KUKA KRL program: EPS_2_25716_MHDR08_A_20251212040354.src

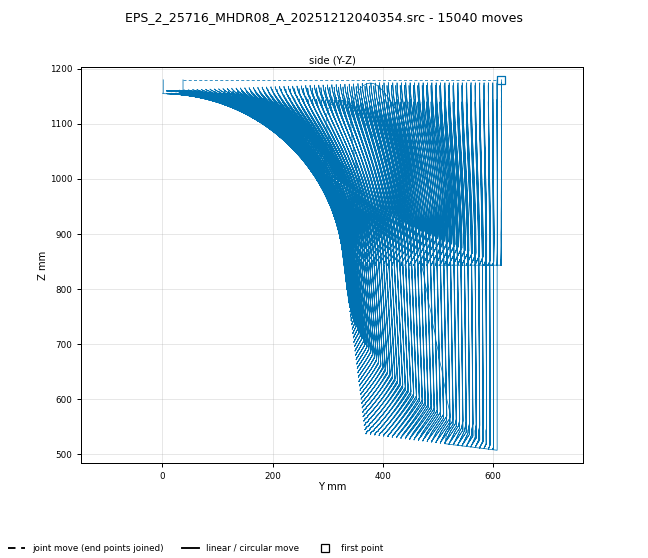
[picture p0: tool path of EPS_2_25716_MHDR08_A_20251212040354.src, 15040 of 15042 moves have a stored position in this frame; points joined in program order, loops and branches not executed]
&ACCESS RVP
&REL 4
&COMMENT QRS 19112012
&PARAM EDITMASK = *
DEF PART()
EXT BAS (BAS_COMMAND :IN,REAL :IN )
INT I
BAS (#INITMOV,0 )

;KUKA QRS Post kuka4.cps  Date:22-06-2017 !

File_ID=2954

QRS_PRE_INIT()

;Init var - Until changes are made in qrs_pre_init
Outlet_Square_prg=0
Inlet_1_Square_prg=0
Inlet_2_Square_prg=0
Inlet_3_Square_prg=0
Inlet_4_Square_prg=0
Inlet_5_Square_prg=0

Outlet_1={X 0.000, Y 400.000, Z 865.000, B 0.000, E1 0.000 }
Inlet_1={X 0.000, Y 400.000, Z 835.000, B 0.000, E1 180.000 }
Outlet_1_type=610
Inlet_1_type=610
;QRS#1=Sidecore dimensions
;QRS#2=600-24" Concrete
;QRS#3=600-24" Concrete
;QRS#4=
;QRS#5=
;QRS#6=
;QRS#7=
;QRS#8=
;QRS#9=S306-34L
;QRS#10=S306-34L
;QRS#11=
;QRS#12=
;QRS#13=
;QRS#14=
;QRS#15=
;QRS#16=1220x127x1524 5'
;QRS#17=EPS Height
;QRS#18=1170
;QRS#19=*
;QRS#20= UPDATED VERSION 22-06-2017
;QRS#21=*
Outlet_Square=0450
Inlet_1_Square=0450
Inlet_2_Square=0
Inlet_3_Square=0
Inlet_4_Square=0
Inlet_5_Square=0
Mill_Square=1
Outlet_Square_Prg=264
Inlet_1_Square_prg=264

QRS_INIT()

$ADVANCE=5

; T1
PTP {E1 172.54,E2 172.54}
PTP {X 0,Y 615.615,A -85,B 0,C 180,E1 172.54,E2 172.54,E3 0,E4 0,E5 0,E6 0}
QRS_SPEED_INIT()
LIN {X 0,Y 615.615,Z 1180,A -85,B 0,C 180,E1 172.54,E2 172.54,E3 0,E4 0,E5 0,E6 0} C_VEL
LIN {X 0,Y 615.615,Z 845.44,A -85,B 0,C 180,E1 172.54,E2 172.54} C_VEL
LIN {X 0,Y 615.56,Z 843.44,A -85,B 0,C 180,E1 172.726,E2 172.726} C_VEL
LIN {X 0,Y 615.848,Z 843.44,A -85,B 0,C 180,E1 176.52,E2 176.52} C_VEL
LIN {X 0,Y 615.869,Z 843.44,A -85,B 0,C 180,E1 181.159,E2 181.159} C_VEL
LIN {X 0,Y 615.847,Z 843.44,A -85,B 0,C 180,E1 185.807,E2 185.807} C_VEL
LIN {X 0,Y 615.82,Z 843.44,A -85,B 0,C 180,E1 190.493,E2 190.493} C_VEL
LIN {X 0,Y 615.8,Z 843.44,A -85,B 0,C 180,E1 195.252,E2 195.252} C_VEL
LIN {X 0,Y 615.797,Z 843.44,A -85,B 0,C 180,E1 200.122,E2 200.122} C_VEL
LIN {X 0,Y 615.751,Z 843.44,A -85,B 0,C 180,E1 205.15,E2 205.15} C_VEL
LIN {X 0,Y 615.231,Z 843.44,A -85,B 0,C 180,E1 207.766,E2 207.766} C_VEL
LIN {X 0,Y 615.751,Z 843.44,A -85,B 0,C 180,E1 210.394,E2 210.394} C_VEL
LIN {X 0,Y 615.134,Z 843.44,A -85,B 0,C 180,E1 213.842,E2 213.842} C_VEL
LIN {X 0,Y 615.66,Z 843.44,A -85,B 0,C 180,E1 215.943,E2 215.943} C_VEL
LIN {X 0,Y 615.4,Z 843.44,A -85,B 0,C 180,E1 217.841,E2 217.841} C_VEL
LIN {X 0,Y 615.353,Z 843.44,A -85,B 0,C 180,E1 218.886,E2 218.886} C_VEL
LIN {X 0,Y 615.632,Z 843.44,A -85,B 0,C 180,E1 221.501,E2 221.501} C_VEL
LIN {X 0,Y 615.673,Z 843.44,A -85,B 0,C 180,E1 225.106,E2 225.106} C_VEL
LIN {X 0,Y 615.248,Z 843.44,A -85,B 0,C 180,E1 228.539,E2 228.539} C_VEL
LIN {X 0,Y 615.62,Z 843.44,A -85,B 0,C 180,E1 231.134,E2 231.134} C_VEL
LIN {X 0,Y 615.854,Z 843.44,A -85,B 0,C 180,E1 236.479,E2 236.479} C_VEL
LIN {X 0,Y 615.651,Z 843.44,A -85,B 0,C 180,E1 236.67,E2 236.67} C_VEL
LIN {X 0,Y 615.102,Z 843.529,A -85,B 0,C 180,E1 236.769,E2 236.769} C_VEL
LIN {X 0,Y 615.262,Z 884.389,A -85,B 0,C 180,E1 237.344,E2 237.344} C_VEL
LIN {X 0,Y 615.454,Z 896.053,A -85,B 0,C 180,E1 237.545,E2 237.545} C_VEL
LIN {X 0,Y 615.368,Z 912.24,A -85,B 0,C 180,E1 237.89,E2 237.89} C_VEL
LIN {X 0,Y 615.486,Z 927.188,A -85,B 0,C 180,E1 238.298,E2 238.298} C_VEL
LIN {X 0,Y 615.404,Z 942.776,A -85,B 0,C 180,E1 238.798,E2 238.798} C_VEL
LIN {X 0,Y 615.565,Z 957.668,A -85,B 0,C 180,E1 239.371,E2 239.371} C_VEL
LIN {X 0,Y 615.586,Z 971.276,A -85,B 0,C 180,E1 239.959,E2 239.959} C_VEL
LIN {X 0,Y 615.496,Z 984.135,A -85,B 0,C 180,E1 240.573,E2 240.573} C_VEL
LIN {X 0,Y 615.632,Z 998.101,A -85,B 0,C 180,E1 241.333,E2 241.333} C_VEL
LIN {X 0,Y 615.649,Z 1011.417,A -85,B 0,C 180,E1 242.129,E2 242.129} C_VEL
LIN {X 0,Y 615.606,Z 1024.492,A -85,B 0,C 180,E1 242.987,E2 242.987} C_VEL
LIN {X 0,Y 615.637,Z 1037.892,A -85,B 0,C 180,E1 243.961,E2 243.961} C_VEL
LIN {X 0,Y 615.676,Z 1049.111,A -85,B 0,C 180,E1 244.847,E2 244.847} C_VEL
LIN {X 0,Y 615.679,Z 1060.739,A -85,B 0,C 180,E1 245.844,E2 245.844} C_VEL
LIN {X 0,Y 615.643,Z 1071.153,A -85,B 0,C 180,E1 246.809,E2 246.809} C_VEL
LIN {X 0,Y 615.684,Z 1081.458,A -85,B 0,C 180,E1 247.846,E2 247.846} C_VEL
LIN {X 0,Y 615.684,Z 1091.552,A -85,B 0,C 180,E1 248.945,E2 248.945} C_VEL
LIN {X 0,Y 615.6,Z 1100.745,A -85,B 0,C 180,E1 250.026,E2 250.026} C_VEL
LIN {X 0,Y 615.667,Z 1109.198,A -85,B 0,C 180,E1 251.104,E2 251.104} C_VEL
LIN {X 0,Y 615.76,Z 1116.662,A -85,B 0,C 180,E1 252.141,E2 252.141} C_VEL
LIN {X 0,Y 615.563,Z 1125.951,A -85,B 0,C 180,E1 253.537,E2 253.537} C_VEL
LIN {X 0,Y 615.67,Z 1133.147,A -85,B 0,C 180,E1 254.744,E2 254.744} C_VEL
LIN {X 0,Y 615.818,Z 1137.992,A -85,B 0,C 180,E1 255.648,E2 255.648} C_VEL
LIN {X 0,Y 615.63,Z 1142.571,A -85,B 0,C 180,E1 256.539,E2 256.539} C_VEL
LIN {X 0,Y 615.562,Z 1146.872,A -85,B 0,C 180,E1 257.431,E2 257.431} C_VEL
LIN {X 0,Y 615.799,Z 1153.082,A -85,B 0,C 180,E1 258.916,E2 258.916} C_VEL
LIN {X 0,Y 615.609,Z 1157.519,A -85,B 0,C 180,E1 260.092,E2 260.092} C_VEL
LIN {X 0,Y 615.522,Z 1161.322,A -85,B 0,C 180,E1 261.266,E2 261.266} C_VEL
LIN {X 0,Y 615.732,Z 1165.013,A -85,B 0,C 180,E1 262.603,E2 262.603} C_VEL
LIN {X 0,Y 615.726,Z 1166.643,A -85,B 0,C 180,E1 263.27,E2 263.27} C_VEL
LIN {X 0,Y 615.525,Z 1168.699,A -85,B 0,C 180,E1 264.19,E2 264.19} C_VEL
LIN {X 0,Y 615.498,Z 1171.145,A -85,B 0,C 180,E1 265.588,E2 265.588} C_VEL
LIN {X 0,Y 615.665,Z 1172.314,A -85,B 0,C 180,E1 266.519,E2 266.519} C_VEL
LIN {X 0,Y 615.731,Z 1173.295,A -85,B 0,C 180,E1 267.448,E2 267.448} C_VEL
LIN {X 0,Y 615.468,Z 1174.226,A -85,B 0,C 180,E1 268.84,E2 268.84} C_VEL
LIN {X 0,Y 615.846,Z 1174.153,A -85,B 0,C 180,E1 271.159,E2 271.159} C_VEL
LIN {X 0,Y 615.739,Z 1173.293,A -85,B 0,C 180,E1 272.552,E2 272.552} C_VEL
LIN {X 0,Y 615.821,Z 1172.284,A -85,B 0,C 180,E1 273.48,E2 273.48} C_VEL
LIN {X 0,Y 615.545,Z 1170.345,A -85,B 0,C 180,E1 274.878,E2 274.878} C_VEL
LIN {X 0,Y 615.53,Z 1168.698,A -85,B 0,C 180,E1 275.81,E2 275.81} C_VEL
LIN {X 0,Y 615.68,Z 1166.586,A -85,B 0,C 180,E1 276.76,E2 276.76} C_VEL
LIN {X 0,Y 615.774,Z 1164.622,A -85,B 0,C 180,E1 277.538,E2 277.538} C_VEL
LIN {X 0,Y 615.541,Z 1161.319,A -85,B 0,C 180,E1 278.733,E2 278.733} C_VEL
LIN {X 0,Y 615.557,Z 1157.527,A -85,B 0,C 180,E1 279.908,E2 279.908} C_VEL
LIN {X 0,Y 615.815,Z 1153.08,A -85,B 0,C 180,E1 281.083,E2 281.083} C_VEL
LIN {X 0,Y 615.534,Z 1146.875,A -85,B 0,C 180,E1 282.57,E2 282.57} C_VEL
LIN {X 0,Y 615.601,Z 1139.632,A -85,B 0,C 180,E1 284.058,E2 284.058} C_VEL
LIN {X 0,Y 615.808,Z 1133.136,A -85,B 0,C 180,E1 285.252,E2 285.252} C_VEL
LIN {X 0,Y 615.58,Z 1124.652,A -85,B 0,C 180,E1 286.664,E2 286.664} C_VEL
LIN {X 0,Y 615.672,Z 1115.983,A -85,B 0,C 180,E1 287.956,E2 287.956} C_VEL
LIN {X 0,Y 615.786,Z 1109.198,A -85,B 0,C 180,E1 288.892,E2 288.892} C_VEL
LIN {X 0,Y 615.593,Z 1098.188,A -85,B 0,C 180,E1 290.283,E2 290.283} C_VEL
LIN {X 0,Y 615.645,Z 1088.781,A -85,B 0,C 180,E1 291.367,E2 291.367} C_VEL
LIN {X 0,Y 615.705,Z 1078.314,A -85,B 0,C 180,E1 292.476,E2 292.476} C_VEL
LIN {X 0,Y 615.619,Z 1068.945,A -85,B 0,C 180,E1 293.404,E2 293.404} C_VEL
LIN {X 0,Y 615.634,Z 1057.804,A -85,B 0,C 180,E1 294.418,E2 294.418} C_VEL
LIN {X 0,Y 615.649,Z 1046.141,A -85,B 0,C 180,E1 295.395,E2 295.395} C_VEL
LIN {X 0,Y 615.633,Z 1033.557,A -85,B 0,C 180,E1 296.362,E2 296.362} C_VEL
LIN {X 0,Y 615.629,Z 1022.093,A -85,B 0,C 180,E1 297.174,E2 297.174} C_VEL
LIN {X 0,Y 615.569,Z 1009.608,A -85,B 0,C 180,E1 297.987,E2 297.987} C_VEL
LIN {X 0,Y 615.637,Z 995.015,A -85,B 0,C 180,E1 298.837,E2 298.837} C_VEL
LIN {X 0,Y 615.587,Z 981.265,A -85,B 0,C 180,E1 299.562,E2 299.562} C_VEL
LIN {X 0,Y 615.487,Z 970.325,A -85,B 0,C 180,E1 300.092,E2 300.092} C_VEL
LIN {X 0,Y 615.592,Z 953.964,A -85,B 0,C 180,E1 300.777,E2 300.777} C_VEL
LIN {X 0,Y 615.412,Z 938.367,A -85,B 0,C 180,E1 301.352,E2 301.352} C_VEL
LIN {X 0,Y 615.482,Z 928.614,A -85,B 0,C 180,E1 301.657,E2 301.657} C_VEL
LIN {X 0,Y 615.497,Z 912.307,A -85,B 0,C 180,E1 302.101,E2 302.101} C_VEL
LIN {X 0,Y 615.3,Z 902.116,A -85,B 0,C 180,E1 302.336,E2 302.336} C_VEL
LIN {X 0,Y 615.425,Z 894.144,A -85,B 0,C 180,E1 302.489,E2 302.489} C_VEL
LIN {X 0,Y 615.395,Z 875.759,A -85,B 0,C 180,E1 302.773,E2 302.773} C_VEL
LIN {X 0,Y 615.134,Z 843.44,A -85,B 0,C 180,E1 303.235,E2 303.235} C_VEL
LIN {X 0,Y 615.646,Z 843.44,A -85,B 0,C 180,E1 303.33,E2 303.33} C_VEL
LIN {X 0,Y 615.853,Z 843.44,A -85,B 0,C 180,E1 303.52,E2 303.52} C_VEL
LIN {X 0,Y 615.62,Z 843.44,A -85,B 0,C 180,E1 308.866,E2 308.866} C_VEL
LIN {X 0,Y 615.242,Z 843.44,A -85,B 0,C 180,E1 311.943,E2 311.943} C_VEL
LIN {X 0,Y 615.68,Z 843.44,A -85,B 0,C 180,E1 314.895,E2 314.895} C_VEL
LIN {X 0,Y 615.622,Z 843.44,A -85,B 0,C 180,E1 318.499,E2 318.499} C_VEL
LIN {X 0,Y 615.342,Z 843.44,A -85,B 0,C 180,E1 321.113,E2 321.113} C_VEL
LIN {X 0,Y 615.398,Z 843.44,A -85,B 0,C 180,E1 322.159,E2 322.159} C_VEL
LIN {X 0,Y 615.655,Z 843.44,A -85,B 0,C 180,E1 324.057,E2 324.057} C_VEL
LIN {X 0,Y 615.136,Z 843.44,A -85,B 0,C 180,E1 326.841,E2 326.841} C_VEL
LIN {X 0,Y 615.745,Z 843.44,A -85,B 0,C 180,E1 329.606,E2 329.606} C_VEL
LIN {X 0,Y 615.22,Z 843.44,A -85,B 0,C 180,E1 332.234,E2 332.234} C_VEL
LIN {X 0,Y 615.744,Z 843.44,A -85,B 0,C 180,E1 334.85,E2 334.85} C_VEL
LIN {X 0,Y 615.807,Z 843.44,A -85,B 0,C 180,E1 339.879,E2 339.879} C_VEL
LIN {X 0,Y 615.814,Z 843.44,A -85,B 0,C 180,E1 343.784,E2 343.784} C_VEL
LIN {X 0,Y 615.822,Z 843.44,A -85,B 0,C 180,E1 349.507,E2 349.507} C_VEL
LIN {X 0,Y 615.852,Z 843.44,A -85,B 0,C 180,E1 354.193,E2 354.193} C_VEL
LIN {X 0,Y 615.873,Z 843.44,A -85,B 0,C 180,E1 358.841,E2 358.841} C_VEL
LIN {X 0,Y 615.858,Z 843.44,A -85,B 0,C 180,E1 363.48,E2 363.48} C_VEL
LIN {X 0,Y 615.852,Z 843.44,A -85,B 0,C 180,E1 368.143,E2 368.143} C_VEL
LIN {X 0,Y 615.792,Z 843.44,A -85,B 0,C 180,E1 372.862,E2 372.862} C_VEL
LIN {X 0,Y 615.794,Z 843.44,A -85,B 0,C 180,E1 377.671,E2 377.671} C_VEL
LIN {X 0,Y 615.796,Z 843.44,A -85,B 0,C 180,E1 377.992,E2 377.992} C_VEL
LIN {X 0,Y 615.771,Z 843.44,A -85,B 0,C 180,E1 382.613,E2 382.613} C_VEL
LIN {X 0,Y 615.222,Z 843.44,A -85,B 0,C 180,E1 385.173,E2 385.173} C_VEL
LIN {X 0,Y 615.721,Z 843.44,A -85,B 0,C 180,E1 387.742,E2 387.742} C_VEL
LIN {X 0,Y 615.236,Z 843.44,A -85,B 0,C 180,E1 390.422,E2 390.422} C_VEL
LIN {X 0,Y 615.867,Z 843.44,A -85,B 0,C 180,E1 393.115,E2 393.115} C_VEL
LIN {X 0,Y 615.552,Z 843.44,A -85,B 0,C 180,E1 395.95,E2 395.95} C_VEL
LIN {X 0,Y 615.615,Z 843.44,A -85,B 0,C 180,E1 397.867,E2 397.867} C_VEL
LIN {X 0,Y 615.605,Z 843.44,A -85,B 0,C 180,E1 401.913,E2 401.913} C_VEL
LIN {X 0,Y 615.188,Z 843.44,A -85,B 0,C 180,E1 405.151,E2 405.151} C_VEL
LIN {X 0,Y 615.672,Z 843.44,A -85,B 0,C 180,E1 408.093,E2 408.093} C_VEL
LIN {X 0,Y 615.538,Z 843.44,A -85,B 0,C 180,E1 412.143,E2 412.143} C_VEL
LIN {X 0,Y 615.49,Z 843.44,A -85,B 0,C 180,E1 414.046,E2 414.046} C_VEL
LIN {X 0,Y 615.859,Z 843.44,A -85,B 0,C 180,E1 416.885,E2 416.885} C_VEL
LIN {X 0,Y 615.114,Z 843.44,A -85,B 0,C 180,E1 417.064,E2 417.064} C_VEL
LIN {X 0,Y 614.862,Z 846.621,A -85,B 0,C 180,E1 417.161,E2 417.161} C_VEL
LIN {X 0,Y 615.416,Z 866.536,A -85,B 0,C 180,E1 417.507,E2 417.507} C_VEL
LIN {X 0,Y 615.402,Z 882.125,A -85,B 0,C 180,E1 417.844,E2 417.844} C_VEL
LIN {X 0,Y 615.386,Z 891.155,A -85,B 0,C 180,E1 418.082,E2 418.082} C_VEL
LIN {X 0,Y 615.464,Z 900.26,A -85,B 0,C 180,E1 418.35,E2 418.35} C_VEL
LIN {X 0,Y 615.435,Z 912.408,A -85,B 0,C 180,E1 418.742,E2 418.742} C_VEL
LIN {X 0,Y 615.43,Z 919.467,A -85,B 0,C 180,E1 419.003,E2 419.003} C_VEL
LIN {X 0,Y 615.562,Z 927.899,A -85,B 0,C 180,E1 419.336,E2 419.336} C_VEL
LIN {X 0,Y 615.593,Z 942.209,A -85,B 0,C 180,E1 419.959,E2 419.959} C_VEL
LIN {X 0,Y 615.496,Z 955.26,A -85,B 0,C 180,E1 420.588,E2 420.588} C_VEL
LIN {X 0,Y 615.62,Z 968.859,A -85,B 0,C 180,E1 421.332,E2 421.332} C_VEL
LIN {X 0,Y 615.633,Z 982.469,A -85,B 0,C 180,E1 422.152,E2 422.152} C_VEL
LIN {X 0,Y 615.603,Z 995.12,A -85,B 0,C 180,E1 422.987,E2 422.987} C_VEL
LIN {X 0,Y 615.636,Z 1007.438,A -85,B 0,C 180,E1 423.88,E2 423.88} C_VEL
LIN {X 0,Y 615.669,Z 1019.641,A -85,B 0,C 180,E1 424.846,E2 424.846} C_VEL
LIN {X 0,Y 615.679,Z 1030.462,A -85,B 0,C 180,E1 425.774,E2 425.774} C_VEL
LIN {X 0,Y 615.64,Z 1041.606,A -85,B 0,C 180,E1 426.809,E2 426.809} C_VEL
LIN {X 0,Y 615.688,Z 1051.876,A -85,B 0,C 180,E1 427.846,E2 427.846} C_VEL
LIN {X 0,Y 615.697,Z 1061.937,A -85,B 0,C 180,E1 428.946,E2 428.946} C_VEL
LIN {X 0,Y 615.595,Z 1071.099,A -85,B 0,C 180,E1 430.026,E2 430.026} C_VEL
LIN {X 0,Y 615.667,Z 1079.523,A -85,B 0,C 180,E1 431.104,E2 431.104} C_VEL
LIN {X 0,Y 615.764,Z 1086.985,A -85,B 0,C 180,E1 432.14,E2 432.14} C_VEL
LIN {X 0,Y 615.566,Z 1096.22,A -85,B 0,C 180,E1 433.537,E2 433.537} C_VEL
LIN {X 0,Y 615.668,Z 1103.4,A -85,B 0,C 180,E1 434.745,E2 434.745} C_VEL
LIN {X 0,Y 615.804,Z 1108.238,A -85,B 0,C 180,E1 435.647,E2 435.647} C_VEL
LIN {X 0,Y 615.627,Z 1112.789,A -85,B 0,C 180,E1 436.539,E2 436.539} C_VEL
LIN {X 0,Y 615.572,Z 1117.063,A -85,B 0,C 180,E1 437.431,E2 437.431} C_VEL
LIN {X 0,Y 615.796,Z 1123.25,A -85,B 0,C 180,E1 438.916,E2 438.916} C_VEL
LIN {X 0,Y 615.603,Z 1127.679,A -85,B 0,C 180,E1 440.092,E2 440.092} C_VEL
LIN {X 0,Y 615.518,Z 1131.468,A -85,B 0,C 180,E1 441.266,E2 441.266} C_VEL
LIN {X 0,Y 615.724,Z 1135.152,A -85,B 0,C 180,E1 442.608,E2 442.608} C_VEL
LIN {X 0,Y 615.727,Z 1136.74,A -85,B 0,C 180,E1 443.27,E2 443.27} C_VEL
LIN {X 0,Y 615.523,Z 1138.799,A -85,B 0,C 180,E1 444.19,E2 444.19} C_VEL
LIN {X 0,Y 615.453,Z 1140.437,A -85,B 0,C 180,E1 445.122,E2 445.122} C_VEL
LIN {X 0,Y 615.677,Z 1142.366,A -85,B 0,C 180,E1 446.519,E2 446.519} C_VEL
LIN {X 0,Y 615.732,Z 1143.326,A -85,B 0,C 180,E1 447.448,E2 447.448} C_VEL
LIN {X 0,Y 615.483,Z 1144.233,A -85,B 0,C 180,E1 448.84,E2 448.84} C_VEL
LIN {X 0,Y 615.843,Z 1144.144,A -85,B 0,C 180,E1 451.159,E2 451.159} C_VEL
LIN {X 0,Y 615.568,Z 1143.294,A -85,B 0,C 180,E1 452.553,E2 452.553} C_VEL
LIN {X 0,Y 615.557,Z 1142.28,A -85,B 0,C 180,E1 453.482,E2 453.482} C_VEL
LIN {X 0,Y 615.709,Z 1141.029,A -85,B 0,C 180,E1 454.411,E2 454.411} C_VEL
LIN {X 0,Y 615.761,Z 1139.446,A -85,B 0,C 180,E1 455.342,E2 455.342} C_VEL
LIN {X 0,Y 615.543,Z 1136.711,A -85,B 0,C 180,E1 456.67,E2 456.67} C_VEL
LIN {X 0,Y 615.605,Z 1133.938,A -85,B 0,C 180,E1 457.76,E2 457.76} C_VEL
LIN {X 0,Y 615.822,Z 1131.13,A -85,B 0,C 180,E1 458.729,E2 458.729} C_VEL
LIN {X 0,Y 615.588,Z 1127.355,A -85,B 0,C 180,E1 459.908,E2 459.908} C_VEL
LIN {X 0,Y 615.554,Z 1121.749,A -85,B 0,C 180,E1 461.384,E2 461.384} C_VEL
LIN {X 0,Y 615.808,Z 1116.642,A -85,B 0,C 180,E1 462.564,E2 462.564} C_VEL
LIN {X 0,Y 615.577,Z 1109.39,A -85,B 0,C 180,E1 464.059,E2 464.059} C_VEL
LIN {X 0,Y 615.62,Z 1102.887,A -85,B 0,C 180,E1 465.257,E2 465.257} C_VEL
LIN {X 0,Y 615.803,Z 1095.663,A -85,B 0,C 180,E1 466.456,E2 466.456} C_VEL
LIN {X 0,Y 615.584,Z 1087.681,A -85,B 0,C 180,E1 467.677,E2 467.677} C_VEL
LIN {X 0,Y 615.634,Z 1077.663,A -85,B 0,C 180,E1 469.05,E2 469.05} C_VEL
LIN {X 0,Y 615.76,Z 1069.127,A -85,B 0,C 180,E1 470.123,E2 470.123} C_VEL
LIN {X 0,Y 615.624,Z 1058.361,A -85,B 0,C 180,E1 471.368,E2 471.368} C_VEL
LIN {X 0,Y 615.652,Z 1049.313,A -85,B 0,C 180,E1 472.334,E2 472.334} C_VEL
LIN {X 0,Y 615.703,Z 1038.425,A -85,B 0,C 180,E1 473.403,E2 473.403} C_VEL
LIN {X 0,Y 615.653,Z 1027.2,A -85,B 0,C 180,E1 474.423,E2 474.423} C_VEL
LIN {X 0,Y 615.64,Z 1015.562,A -85,B 0,C 180,E1 475.395,E2 475.395} C_VEL
LIN {X 0,Y 615.649,Z 1004.057,A -85,B 0,C 180,E1 476.281,E2 476.281} C_VEL
LIN {X 0,Y 615.649,Z 991.401,A -85,B 0,C 180,E1 477.174,E2 477.174} C_VEL
LIN {X 0,Y 615.626,Z 978.933,A -85,B 0,C 180,E1 477.98,E2 477.98} C_VEL
LIN {X 0,Y 615.59,Z 967.05,A -85,B 0,C 180,E1 478.685,E2 478.685} C_VEL
LIN {X 0,Y 615.616,Z 951.527,A -85,B 0,C 180,E1 479.503,E2 479.503} C_VEL
LIN {X 0,Y 615.48,Z 938.091,A -85,B 0,C 180,E1 480.146,E2 480.146} C_VEL
LIN {X 0,Y 615.584,Z 924.036,A -85,B 0,C 180,E1 480.73,E2 480.73} C_VEL
LIN {X 0,Y 615.577,Z 908.655,A -85,B 0,C 180,E1 481.288,E2 481.288} C_VEL
LIN {X 0,Y 615.335,Z 894.951,A -85,B 0,C 180,E1 481.731,E2 481.731} C_VEL
LIN {X 0,Y 615.584,Z 879.877,A -85,B 0,C 180,E1 482.109,E2 482.109} C_VEL
LIN {X 0,Y 615.542,Z 864.831,A -85,B 0,C 180,E1 482.426,E2 482.426} C_VEL
LIN {X 0,Y 615.35,Z 855.68,A -85,B 0,C 180,E1 482.585,E2 482.585} C_VEL
LIN {X 0,Y 614.951,Z 848.797,A -85,B 0,C 180,E1 482.714,E2 482.714} C_VEL
LIN {X 0,Y 614.443,Z 845.073,A -85,B 0,C 180,E1 482.795,E2 482.795} C_VEL
LIN {X 0,Y 614.72,Z 843.44,A -85,B 0,C 180,E1 482.88,E2 482.88} C_VEL
LIN {X 0,Y 615.865,Z 843.44,A -85,B 0,C 180,E1 483.115,E2 483.115} C_VEL
LIN {X 0,Y 615.646,Z 843.44,A -85,B 0,C 180,E1 483.913,E2 483.913} C_VEL
LIN {X 0,Y 615.593,Z 843.44,A -85,B 0,C 180,E1 488.868,E2 488.868} C_VEL
LIN {X 0,Y 615.221,Z 843.44,A -85,B 0,C 180,E1 491.945,E2 491.945} C_VEL
LIN {X 0,Y 615.662,Z 843.44,A -85,B 0,C 180,E1 494.893,E2 494.893} C_VEL
LIN {X 0,Y 615.623,Z 843.44,A -85,B 0,C 180,E1 498.499,E2 498.499} C_VEL
LIN {X 0,Y 615.338,Z 843.44,A -85,B 0,C 180,E1 501.113,E2 501.113} C_VEL
LIN {X 0,Y 615.38,Z 843.44,A -85,B 0,C 180,E1 502.162,E2 502.162} C_VEL
LIN {X 0,Y 615.647,Z 843.44,A -85,B 0,C 180,E1 504.056,E2 504.056} C_VEL
LIN {X 0,Y 615.135,Z 843.44,A -85,B 0,C 180,E1 506.841,E2 506.841} C_VEL
LIN {X 0,Y 615.75,Z 843.44,A -85,B 0,C 180,E1 509.606,E2 509.606} C_VEL
LIN {X 0,Y 615.222,Z 843.44,A -85,B 0,C 180,E1 512.234,E2 512.234} C_VEL
LIN {X 0,Y 615.735,Z 843.44,A -85,B 0,C 180,E1 514.849,E2 514.849} C_VEL
LIN {X 0,Y 615.818,Z 843.44,A -85,B 0,C 180,E1 519.879,E2 519.879} C_VEL
LIN {X 0,Y 615.53,Z 843.44,A -85,B 0,C 180,E1 522.322,E2 522.322} C_VEL
LIN {X 0,Y 615.632,Z 843.44,A -85,B 0,C 180,E1 524.743,E2 524.743} C_VEL
LIN {X 0,Y 615.802,Z 843.44,A -85,B 0,C 180,E1 527.138,E2 527.138} C_VEL
LIN {X 0,Y 615.859,Z 843.44,A -85,B 0,C 180,E1 531.857,E2 531.857} C_VEL
LIN {X 0,Y 615.56,Z 843.44,A -85,B 0,C 180,E1 532.726,E2 532.726} C_VEL
LIN {X 0,Y 611.541,Z 843.44,A -85,B 0,C 180,E1 534.313,E2 534.313} C_VEL
LIN {X 0,Y 607.674,Z 843.44,A -85,B 0,C 180,E1 535.921,E2 535.921} C_VEL
LIN {X 0,Y 607.881,Z 843.44,A -85,B 0,C 180,E1 541.423,E2 541.423} C_VEL
LIN {X 0,Y 607.65,Z 843.44,A -85,B 0,C 180,E1 546.615,E2 546.615} C_VEL
LIN {X 0,Y 607.601,Z 843.44,A -85,B 0,C 180,E1 551.46,E2 551.46} C_VEL
LIN {X 0,Y 607.656,Z 843.44,A -85,B 0,C 180,E1 555.852,E2 555.852} C_VEL
LIN {X 0,Y 607.803,Z 843.44,A -85,B 0,C 180,E1 560.339,E2 560.339} C_VEL
LIN {X 0,Y 607.775,Z 843.44,A -85,B 0,C 180,E1 564.965,E2 564.965} C_VEL
LIN {X 0,Y 607.621,Z 843.44,A -85,B 0,C 180,E1 569.78,E2 569.78} C_VEL
LIN {X 0,Y 607.6,Z 843.44,A -85,B 0,C 180,E1 576.586,E2 576.586} C_VEL
LIN {X 0,Y 607.592,Z 843.44,A -85,B 0,C 180,E1 582.109,E2 582.109} C_VEL
LIN {X 0,Y 607.447,Z 843.44,A -85,B 0,C 180,E1 586.087,E2 586.087} C_VEL
LIN {X 0,Y 607.547,Z 843.44,A -85,B 0,C 180,E1 591.615,E2 591.615} C_VEL
LIN {X 0,Y 607.882,Z 843.44,A -85,B 0,C 180,E1 596.309,E2 596.309} C_VEL
LIN {X 0,Y 608.694,Z 910.185,A -85,B 0,C 180,E1 597.444,E2 597.444} C_VEL
LIN {X 0,Y 608.624,Z 952.563,A -85,B 0,C 180,E1 598.779,E2 598.779} C_VEL
LIN {X 0,Y 608.455,Z 992.837,A -85,B 0,C 180,E1 600.672,E2 600.672} C_VEL
LIN {X 0,Y 608.284,Z 1030.382,A -85,B 0,C 180,E1 603.064,E2 603.064} C_VEL
LIN {X 0,Y 608.152,Z 1064.017,A -85,B 0,C 180,E1 605.832,E2 605.832} C_VEL
LIN {X 0,Y 608.002,Z 1093.584,A -85,B 0,C 180,E1 608.907,E2 608.907} C_VEL
LIN {X 0,Y 607.946,Z 1119.324,A -85,B 0,C 180,E1 612.298,E2 612.298} C_VEL
LIN {X 0,Y 607.917,Z 1140.95,A -85,B 0,C 180,E1 615.994,E2 615.994} C_VEL
LIN {X 0,Y 607.762,Z 1157.905,A -85,B 0,C 180,E1 619.991,E2 619.991} C_VEL
LIN {X 0,Y 607.765,Z 1167.962,A -85,B 0,C 180,E1 623.584,E2 623.584} C_VEL
LIN {X 0,Y 607.833,Z 1173.637,A -85,B 0,C 180,E1 627.154,E2 627.154} C_VEL
LIN {X 0,Y 607.927,Z 1174.659,A -85,B 0,C 180,E1 631.423,E2 631.423} C_VEL
LIN {X 0,Y 607.66,Z 1170.729,A -85,B 0,C 180,E1 634.986,E2 634.986} C_VEL
LIN {X 0,Y 607.708,Z 1162.531,A -85,B 0,C 180,E1 638.568,E2 638.568} C_VEL
LIN {X 0,Y 607.717,Z 1149.388,A -85,B 0,C 180,E1 642.185,E2 642.185} C_VEL
LIN {X 0,Y 607.894,Z 1130.904,A -85,B 0,C 180,E1 645.847,E2 645.847} C_VEL
LIN {X 0,Y 607.971,Z 1107.131,A -85,B 0,C 180,E1 649.414,E2 649.414} C_VEL
LIN {X 0,Y 608.103,Z 1077.903,A -85,B 0,C 180,E1 652.814,E2 652.814} C_VEL
LIN {X 0,Y 608.241,Z 1044.822,A -85,B 0,C 180,E1 655.831,E2 655.831} C_VEL
LIN {X 0,Y 608.39,Z 1008.415,A -85,B 0,C 180,E1 658.419,E2 658.419} C_VEL
LIN {X 0,Y 608.572,Z 967.8,A -85,B 0,C 180,E1 660.583,E2 660.583} C_VEL
LIN {X 0,Y 608.756,Z 925.8,A -85,B 0,C 180,E1 662.137,E2 662.137} C_VEL
LIN {X 0,Y 608.78,Z 887.562,A -85,B 0,C 180,E1 662.996,E2 662.996} C_VEL
LIN {X 0,Y 607.881,Z 843.44,A -85,B 0,C 180,E1 663.693,E2 663.693} C_VEL
LIN {X 0,Y 607.456,Z 843.44,A -85,B 0,C 180,E1 669.641,E2 669.641} C_VEL
LIN {X 0,Y 607.521,Z 843.44,A -85,B 0,C 180,E1 675.936,E2 675.936} C_VEL
LIN {X 0,Y 607.417,Z 843.44,A -85,B 0,C 180,E1 680.366,E2 680.366} C_VEL
LIN {X 0,Y 607.4,Z 843.44,A -85,B 0,C 180,E1 685.153,E2 685.153} C_VEL
LIN {X 0,Y 607.567,Z 843.44,A -85,B 0,C 180,E1 690.377,E2 690.377} C_VEL
LIN {X 0,Y 607.782,Z 843.44,A -85,B 0,C 180,E1 695.035,E2 695.035} C_VEL
LIN {X 0,Y 607.676,Z 843.44,A -85,B 0,C 180,E1 700.672,E2 700.672} C_VEL
LIN {X 0,Y 607.276,Z 843.44,A -85,B 0,C 180,E1 705.612,E2 705.612} C_VEL
LIN {X 0,Y 607.749,Z 843.44,A -85,B 0,C 180,E1 709.991,E2 709.991} C_VEL
LIN {X 0,Y 607.925,Z 843.44,A -85,B 0,C 180,E1 714.302,E2 714.302} C_VEL
LIN {X 0,Y 607.59,Z 843.44,A -85,B 0,C 180,E1 720,E2 720} C_VEL
LIN {X 0,Y 607.669,Z 843.44,A -85,B 0,C 180,E1 724.272,E2 724.272} C_VEL
LIN {X 0,Y 607.799,Z 843.44,A -85,B 0,C 180,E1 728.566,E2 728.566} C_VEL
LIN {X 0,Y 607.865,Z 843.44,A -85,B 0,C 180,E1 732.91,E2 732.91} C_VEL
LIN {X 0,Y 607.592,Z 843.44,A -85,B 0,C 180,E1 738.836,E2 738.836} C_VEL
LIN {X 0,Y 607.584,Z 843.44,A -85,B 0,C 180,E1 743.413,E2 743.413} C_VEL
LIN {X 0,Y 607.668,Z 843.44,A -85,B 0,C 180,E1 748.151,E2 748.151} C_VEL
LIN {X 0,Y 607.956,Z 843.44,A -85,B 0,C 180,E1 753.096,E2 753.096} C_VEL
LIN {X 0,Y 607.561,Z 843.44,A -85,B 0,C 180,E1 758.382,E2 758.382} C_VEL
LIN {X 0,Y 607.634,Z 843.44,A -85,B 0,C 180,E1 762.105,E2 762.105} C_VEL
LIN {X 0,Y 607.753,Z 843.44,A -85,B 0,C 180,E1 768.146,E2 768.146} C_VEL
LIN {X 0,Y 607.557,Z 843.44,A -85,B 0,C 180,E1 773.409,E2 773.409} C_VEL
LIN {X 0,Y 607.902,Z 843.44,A -85,B 0,C 180,E1 776.687,E2 776.687} C_VEL
LIN {X 0,Y 608.629,Z 889.434,A -85,B 0,C 180,E1 777.639,E2 777.639} C_VEL
LIN {X 0,Y 608.621,Z 928.772,A -85,B 0,C 180,E1 778.986,E2 778.986} C_VEL
LIN {X 0,Y 608.5,Z 967.382,A -85,B 0,C 180,E1 780.877,E2 780.877} C_VEL
LIN {X 0,Y 608.281,Z 1006.644,A -85,B 0,C 180,E1 783.478,E2 783.478} C_VEL
LIN {X 0,Y 608.106,Z 1040.694,A -85,B 0,C 180,E1 786.413,E2 786.413} C_VEL
LIN {X 0,Y 607.909,Z 1070.334,A -85,B 0,C 180,E1 789.664,E2 789.664} C_VEL
LIN {X 0,Y 607.792,Z 1095.675,A -85,B 0,C 180,E1 793.224,E2 793.224} C_VEL
LIN {X 0,Y 607.753,Z 1114.665,A -85,B 0,C 180,E1 796.722,E2 796.722} C_VEL
LIN {X 0,Y 607.705,Z 1129.227,A -85,B 0,C 180,E1 800.351,E2 800.351} C_VEL
LIN {X 0,Y 607.76,Z 1138.059,A -85,B 0,C 180,E1 803.584,E2 803.584} C_VEL
LIN {X 0,Y 607.844,Z 1143.679,A -85,B 0,C 180,E1 807.154,E2 807.154} C_VEL
LIN {X 0,Y 607.892,Z 1144.632,A -85,B 0,C 180,E1 811.422,E2 811.422} C_VEL
LIN {X 0,Y 607.833,Z 1139.424,A -85,B 0,C 180,E1 815.699,E2 815.699} C_VEL
LIN {X 0,Y 607.755,Z 1128.941,A -85,B 0,C 180,E1 819.648,E2 819.648} C_VEL
LIN {X 0,Y 607.83,Z 1114.235,A -85,B 0,C 180,E1 823.276,E2 823.276} C_VEL
LIN {X 0,Y 607.912,Z 1093.883,A -85,B 0,C 180,E1 826.958,E2 826.958} C_VEL
LIN {X 0,Y 608.023,Z 1068.024,A -85,B 0,C 180,E1 830.521,E2 830.521} C_VEL
LIN {X 0,Y 608.144,Z 1037.706,A -85,B 0,C 180,E1 833.779,E2 833.779} C_VEL
LIN {X 0,Y 608.303,Z 1004.165,A -85,B 0,C 180,E1 836.616,E2 836.616} C_VEL
LIN {X 0,Y 608.477,Z 965.756,A -85,B 0,C 180,E1 839.124,E2 839.124} C_VEL
LIN {X 0,Y 608.683,Z 925.47,A -85,B 0,C 180,E1 841.062,E2 841.062} C_VEL
LIN {X 0,Y 608.784,Z 885.127,A -85,B 0,C 180,E1 842.377,E2 842.377} C_VEL
LIN {X 0,Y 607.891,Z 843.44,A -85,B 0,C 180,E1 843.261,E2 843.261} C_VEL
LIN {X 0,Y 607.459,Z 843.44,A -85,B 0,C 180,E1 849.642,E2 849.642} C_VEL
LIN {X 0,Y 607.512,Z 843.44,A -85,B 0,C 180,E1 855.935,E2 855.935} C_VEL
LIN {X 0,Y 607.389,Z 843.44,A -85,B 0,C 180,E1 860.369,E2 860.369} C_VEL
LIN {X 0,Y 607.389,Z 843.44,A -85,B 0,C 180,E1 865.153,E2 865.153} C_VEL
LIN {X 0,Y 607.558,Z 843.44,A -85,B 0,C 180,E1 870.378,E2 870.378} C_VEL
LIN {X 0,Y 607.76,Z 843.44,A -85,B 0,C 180,E1 875.034,E2 875.034} C_VEL
LIN {X 0,Y 607.658,Z 843.44,A -85,B 0,C 180,E1 881.167,E2 881.167} C_VEL
LIN {X 0,Y 607.905,Z 843.44,A -85,B 0,C 180,E1 887.091,E2 887.091} C_VEL
LIN {X 0,Y 607.627,Z 843.44,A -85,B 0,C 180,E1 892.867,E2 892.867} C_VEL
LIN {X 0,Y 607.674,Z 843.44,A -85,B 0,C 180,E1 895.921,E2 895.921} C_VEL
LIN {X 0,Y 606.348,Z 843.44,A -85,B 0,C 180,E1 896.734,E2 896.734} C_VEL
LIN {X 0,Y 599.658,Z 843.44,A -85,B 0,C 180,E1 898.945,E2 898.945} C_VEL
LIN {X 0,Y 599.58,Z 843.44,A -85,B 0,C 180,E1 899.154,E2 899.154} C_VEL
LIN {X 0,Y 599.632,Z 843.44,A -85,B 0,C 180,E1 902.885,E2 902.885} C_VEL
LIN {X 0,Y 599.609,Z 843.44,A -85,B 0,C 180,E1 907.229,E2 907.229} C_VEL
LIN {X 0,Y 599.658,Z 843.44,A -85,B 0,C 180,E1 911.614,E2 911.614} C_VEL
LIN {X 0,Y 599.504,Z 843.44,A -85,B 0,C 180,E1 916.962,E2 916.962} C_VEL
LIN {X 0,Y 599.567,Z 843.44,A -85,B 0,C 180,E1 921.373,E2 921.373} C_VEL
LIN {X 0,Y 599.781,Z 843.44,A -85,B 0,C 180,E1 925.321,E2 925.321} C_VEL
LIN {X 0,Y 599.535,Z 843.44,A -85,B 0,C 180,E1 931.155,E2 931.155} C_VEL
LIN {X 0,Y 599.634,Z 843.44,A -85,B 0,C 180,E1 937.153,E2 937.153} C_VEL
LIN {X 0,Y 599.567,Z 843.44,A -85,B 0,C 180,E1 943.123,E2 943.123} C_VEL
LIN {X 0,Y 599.395,Z 843.44,A -85,B 0,C 180,E1 949.113,E2 949.113} C_VEL
LIN {X 0,Y 599.29,Z 843.44,A -85,B 0,C 180,E1 953.681,E2 953.681} C_VEL
LIN {X 0,Y 599.786,Z 844.081,A -85,B 0,C 180,E1 955.813,E2 955.813} C_VEL
LIN {X 0,Y 601.916,Z 849.342,A -85,B 0,C 180,E1 956.025,E2 956.025} C_VEL
LIN {X 0,Y 602.01,Z 910.186,A -85,B 0,C 180,E1 957.037,E2 957.037} C_VEL
LIN {X 0,Y 601.759,Z 952.017,A -85,B 0,C 180,E1 958.361,E2 958.361} C_VEL
LIN {X 0,Y 601.366,Z 991.871,A -85,B 0,C 180,E1 960.238,E2 960.238} C_VEL
LIN {X 0,Y 601.011,Z 1029.073,A -85,B 0,C 180,E1 962.614,E2 962.614} C_VEL
LIN {X 0,Y 600.698,Z 1062.974,A -85,B 0,C 180,E1 965.414,E2 965.414} C_VEL
LIN {X 0,Y 600.345,Z 1093.078,A -85,B 0,C 180,E1 968.564,E2 968.564} C_VEL
LIN {X 0,Y 600.21,Z 1119.326,A -85,B 0,C 180,E1 972.062,E2 972.062} C_VEL
LIN {X 0,Y 600.11,Z 1140.952,A -85,B 0,C 180,E1 975.808,E2 975.808} C_VEL
LIN {X 0,Y 599.883,Z 1157.905,A -85,B 0,C 180,E1 979.858,E2 979.858} C_VEL
LIN {X 0,Y 599.905,Z 1167.736,A -85,B 0,C 180,E1 983.395,E2 983.395} C_VEL
LIN {X 0,Y 599.932,Z 1173.637,A -85,B 0,C 180,E1 987.117,E2 987.117} C_VEL
LIN {X 0,Y 600.024,Z 1174.659,A -85,B 0,C 180,E1 991.441,E2 991.441} C_VEL
LIN {X 0,Y 599.765,Z 1170.729,A -85,B 0,C 180,E1 995.052,E2 995.052} C_VEL
LIN {X 0,Y 599.802,Z 1162.531,A -85,B 0,C 180,E1 998.682,E2 998.682} C_VEL
LIN {X 0,Y 599.852,Z 1149.389,A -85,B 0,C 180,E1 1002.347,E2 1002.347} C_VEL
LIN {X 0,Y 600.036,Z 1130.906,A -85,B 0,C 180,E1 1006.06,E2 1006.06} C_VEL
LIN {X 0,Y 600.226,Z 1107.133,A -85,B 0,C 180,E1 1009.675,E2 1009.675} C_VEL
LIN {X 0,Y 600.494,Z 1077.548,A -85,B 0,C 180,E1 1013.156,E2 1013.156} C_VEL
LIN {X 0,Y 600.864,Z 1044.824,A -85,B 0,C 180,E1 1016.172,E2 1016.172} C_VEL
LIN {X 0,Y 601.249,Z 1008.43,A -85,B 0,C 180,E1 1018.787,E2 1018.787} C_VEL
LIN {X 0,Y 601.651,Z 967.745,A -85,B 0,C 180,E1 1020.976,E2 1020.976} C_VEL
LIN {X 0,Y 602.033,Z 926.243,A -85,B 0,C 180,E1 1022.526,E2 1022.526} C_VEL
LIN {X 0,Y 602.164,Z 886.287,A -85,B 0,C 180,E1 1023.427,E2 1023.427} C_VEL
LIN {X 0,Y 601.425,Z 848.23,A -85,B 0,C 180,E1 1024.022,E2 1024.022} C_VEL
LIN {X 0,Y 599.715,Z 843.44,A -85,B 0,C 180,E1 1024.279,E2 1024.279} C_VEL
LIN {X 0,Y 599.585,Z 843.44,A -85,B 0,C 180,E1 1028.991,E2 1028.991} C_VEL
LIN {X 0,Y 599.539,Z 843.44,A -85,B 0,C 180,E1 1035.193,E2 1035.193} C_VEL
LIN {X 0,Y 599.518,Z 843.44,A -85,B 0,C 180,E1 1041.006,E2 1041.006} C_VEL
LIN {X 0,Y 599.543,Z 843.44,A -85,B 0,C 180,E1 1044.629,E2 1044.629} C_VEL
LIN {X 0,Y 599.63,Z 843.44,A -85,B 0,C 180,E1 1049.782,E2 1049.782} C_VEL
LIN {X 0,Y 599.855,Z 843.44,A -85,B 0,C 180,E1 1054.908,E2 1054.908} C_VEL
LIN {X 0,Y 599.75,Z 843.44,A -85,B 0,C 180,E1 1060.908,E2 1060.908} C_VEL
LIN {X 0,Y 599.412,Z 843.44,A -85,B 0,C 180,E1 1065.419,E2 1065.419} C_VEL
LIN {X 0,Y 599.809,Z 843.44,A -85,B 0,C 180,E1 1069.857,E2 1069.857} C_VEL
LIN {X 0,Y 600.021,Z 843.44,A -85,B 0,C 180,E1 1074.227,E2 1074.227} C_VEL
LIN {X 0,Y 599.689,Z 843.44,A -85,B 0,C 180,E1 1080,E2 1080} C_VEL
LIN {X 0,Y 599.753,Z 843.44,A -85,B 0,C 180,E1 1084.329,E2 1084.329} C_VEL
LIN {X 0,Y 599.852,Z 843.44,A -85,B 0,C 180,E1 1088.681,E2 1088.681} C_VEL
LIN {X 0,Y 599.887,Z 843.44,A -85,B 0,C 180,E1 1093.084,E2 1093.084} C_VEL
LIN {X 0,Y 599.654,Z 843.44,A -85,B 0,C 180,E1 1099.094,E2 1099.094} C_VEL
LIN {X 0,Y 599.589,Z 843.44,A -85,B 0,C 180,E1 1103.745,E2 1103.745} C_VEL
LIN {X 0,Y 599.67,Z 843.44,A -85,B 0,C 180,E1 1108.561,E2 1108.561} C_VEL
LIN {X 0,Y 599.837,Z 843.44,A -85,B 0,C 180,E1 1113.882,E2 1113.882} C_VEL
LIN {X 0,Y 599.519,Z 843.44,A -85,B 0,C 180,E1 1118.994,E2 1118.994} C_VEL
LIN {X 0,Y 599.435,Z 843.44,A -85,B 0,C 180,E1 1123.11,E2 1123.11} C_VEL
LIN {X 0,Y 599.549,Z 843.44,A -85,B 0,C 180,E1 1129.126,E2 1129.126} C_VEL
LIN {X 0,Y 599.631,Z 843.44,A -85,B 0,C 180,E1 1134.633,E2 1134.633} C_VEL
LIN {X 0,Y 599.854,Z 843.861,A -85,B 0,C 180,E1 1136.194,E2 1136.194} C_VEL
LIN {X 0,Y 601.737,Z 851.656,A -85,B 0,C 180,E1 1136.424,E2 1136.424} C_VEL
LIN {X 0,Y 601.918,Z 897.01,A -85,B 0,C 180,E1 1137.447,E2 1137.447} C_VEL
LIN {X 0,Y 601.697,Z 937.866,A -85,B 0,C 180,E1 1138.987,E2 1138.987} C_VEL
LIN {X 0,Y 601.301,Z 975.81,A -85,B 0,C 180,E1 1141.01,E2 1141.01} C_VEL
LIN {X 0,Y 600.896,Z 1011.638,A -85,B 0,C 180,E1 1143.528,E2 1143.528} C_VEL
LIN {X 0,Y 600.492,Z 1044.635,A -85,B 0,C 180,E1 1146.501,E2 1146.501} C_VEL
LIN {X 0,Y 600.192,Z 1072.155,A -85,B 0,C 180,E1 1149.63,E2 1149.63} C_VEL
LIN {X 0,Y 600.002,Z 1096.464,A -85,B 0,C 180,E1 1153.133,E2 1153.133} C_VEL
LIN {X 0,Y 599.878,Z 1116.414,A -85,B 0,C 180,E1 1156.915,E2 1156.915} C_VEL
LIN {X 0,Y 599.78,Z 1130.376,A -85,B 0,C 180,E1 1160.588,E2 1160.588} C_VEL
LIN {X 0,Y 599.752,Z 1139.6,A -85,B 0,C 180,E1 1164.224,E2 1164.224} C_VEL
LIN {X 0,Y 599.942,Z 1143.678,A -85,B 0,C 180,E1 1167.116,E2 1167.116} C_VEL
LIN {X 0,Y 599.986,Z 1144.632,A -85,B 0,C 180,E1 1171.441,E2 1171.441} C_VEL
LIN {X 0,Y 599.944,Z 1139.426,A -85,B 0,C 180,E1 1175.774,E2 1175.774} C_VEL
LIN {X 0,Y 599.852,Z 1128.943,A -85,B 0,C 180,E1 1179.776,E2 1179.776} C_VEL
LIN {X 0,Y 599.965,Z 1114.294,A -85,B 0,C 180,E1 1183.442,E2 1183.442} C_VEL
LIN {X 0,Y 600.078,Z 1094.13,A -85,B 0,C 180,E1 1187.149,E2 1187.149} C_VEL
LIN {X 0,Y 600.334,Z 1067.642,A -85,B 0,C 180,E1 1190.843,E2 1190.843} C_VEL
LIN {X 0,Y 600.633,Z 1036.688,A -85,B 0,C 180,E1 1194.192,E2 1194.192} C_VEL
LIN {X 0,Y 601.026,Z 1002.372,A -85,B 0,C 180,E1 1197.097,E2 1197.097} C_VEL
LIN {X 0,Y 601.407,Z 965.181,A -85,B 0,C 180,E1 1199.532,E2 1199.532} C_VEL
LIN {X 0,Y 601.832,Z 925.606,A -85,B 0,C 180,E1 1201.451,E2 1201.451} C_VEL
LIN {X 0,Y 602.055,Z 886.928,A -85,B 0,C 180,E1 1202.736,E2 1202.736} C_VEL
LIN {X 0,Y 601.053,Z 847.487,A -85,B 0,C 180,E1 1203.589,E2 1203.589} C_VEL
LIN {X 0,Y 599.874,Z 843.44,A -85,B 0,C 180,E1 1203.764,E2 1203.764} C_VEL
LIN {X 0,Y 599.544,Z 843.44,A -85,B 0,C 180,E1 1208.994,E2 1208.994} C_VEL
LIN {X 0,Y 599.527,Z 843.44,A -85,B 0,C 180,E1 1215.192,E2 1215.192} C_VEL
LIN {X 0,Y 599.499,Z 843.44,A -85,B 0,C 180,E1 1221.005,E2 1221.005} C_VEL
LIN {X 0,Y 599.522,Z 843.44,A -85,B 0,C 180,E1 1224.627,E2 1224.627} C_VEL
LIN {X 0,Y 599.627,Z 843.44,A -85,B 0,C 180,E1 1229.782,E2 1229.782} C_VEL
LIN {X 0,Y 599.814,Z 843.44,A -85,B 0,C 180,E1 1234.916,E2 1234.916} C_VEL
LIN {X 0,Y 599.791,Z 843.44,A -85,B 0,C 180,E1 1240.91,E2 1240.91} C_VEL
LIN {X 0,Y 599.958,Z 843.44,A -85,B 0,C 180,E1 1246.917,E2 1246.917} C_VEL
LIN {X 0,Y 599.728,Z 843.44,A -85,B 0,C 180,E1 1252.773,E2 1252.773} C_VEL
LIN {X 0,Y 599.832,Z 843.44,A -85,B 0,C 180,E1 1257.116,E2 1257.116} C_VEL
LIN {X 0,Y 599.58,Z 843.44,A -85,B 0,C 180,E1 1259.154,E2 1259.154} C_VEL
LIN {X 0,Y 598.416,Z 843.44,A -85,B 0,C 180,E1 1259.983,E2 1259.983} C_VEL
LIN {X 0,Y 591.792,Z 843.44,A -85,B 0,C 180,E1 1262.451,E2 1262.451} C_VEL
LIN {X 0,Y 591.702,Z 843.44,A -85,B 0,C 180,E1 1267.326,E2 1267.326} C_VEL
LIN {X 0,Y 591.721,Z 843.44,A -85,B 0,C 180,E1 1271.772,E2 1271.772} C_VEL
LIN {X 0,Y 591.747,Z 843.44,A -85,B 0,C 180,E1 1276.29,E2 1276.29} C_VEL
LIN {X 0,Y 591.801,Z 843.44,A -85,B 0,C 180,E1 1280.914,E2 1280.914} C_VEL
LIN {X 0,Y 591.637,Z 843.44,A -85,B 0,C 180,E1 1286.786,E2 1286.786} C_VEL
LIN {X 0,Y 591.661,Z 843.44,A -85,B 0,C 180,E1 1290.669,E2 1290.669} C_VEL
LIN {X 0,Y 591.692,Z 843.44,A -85,B 0,C 180,E1 1295.913,E2 1295.913} C_VEL
LIN {X 0,Y 591.635,Z 843.44,A -85,B 0,C 180,E1 1301.539,E2 1301.539} C_VEL
LIN {X 0,Y 591.494,Z 843.44,A -85,B 0,C 180,E1 1306.463,E2 1306.463} C_VEL
LIN {X 0,Y 591.5,Z 843.44,A -85,B 0,C 180,E1 1312.263,E2 1312.263} C_VEL
LIN {X 0,Y 591.661,Z 843.44,A -85,B 0,C 180,E1 1315.243,E2 1315.243} C_VEL
LIN {X 0,Y 595.371,Z 852.197,A -85,B 0,C 180,E1 1315.64,E2 1315.64} C_VEL
LIN {X 0,Y 595.367,Z 910.414,A -85,B 0,C 180,E1 1316.626,E2 1316.626} C_VEL
LIN {X 0,Y 594.917,Z 953.682,A -85,B 0,C 180,E1 1318.018,E2 1318.018} C_VEL
LIN {X 0,Y 594.299,Z 995.331,A -85,B 0,C 180,E1 1320.041,E2 1320.041} C_VEL
LIN {X 0,Y 593.697,Z 1034.855,A -85,B 0,C 180,E1 1322.68,E2 1322.68} C_VEL
LIN {X 0,Y 593.093,Z 1070.457,A -85,B 0,C 180,E1 1325.8,E2 1325.8} C_VEL
LIN {X 0,Y 592.534,Z 1101.391,A -85,B 0,C 180,E1 1329.298,E2 1329.298} C_VEL
LIN {X 0,Y 592.205,Z 1126.755,A -85,B 0,C 180,E1 1333,E2 1333} C_VEL
LIN {X 0,Y 592.048,Z 1146.204,A -85,B 0,C 180,E1 1336.739,E2 1336.739} C_VEL
LIN {X 0,Y 591.921,Z 1160.236,A -85,B 0,C 180,E1 1340.462,E2 1340.462} C_VEL
LIN {X 0,Y 591.879,Z 1169.517,A -85,B 0,C 180,E1 1344.147,E2 1344.147} C_VEL
LIN {X 0,Y 592.021,Z 1173.637,A -85,B 0,C 180,E1 1347.078,E2 1347.078} C_VEL
LIN {X 0,Y 592.121,Z 1174.659,A -85,B 0,C 180,E1 1351.46,E2 1351.46} C_VEL
LIN {X 0,Y 591.877,Z 1170.73,A -85,B 0,C 180,E1 1355.12,E2 1355.12} C_VEL
LIN {X 0,Y 591.905,Z 1162.531,A -85,B 0,C 180,E1 1358.799,E2 1358.799} C_VEL
LIN {X 0,Y 591.984,Z 1149.39,A -85,B 0,C 180,E1 1362.514,E2 1362.514} C_VEL
LIN {X 0,Y 592.204,Z 1130.907,A -85,B 0,C 180,E1 1366.278,E2 1366.278} C_VEL
LIN {X 0,Y 592.506,Z 1106.845,A -85,B 0,C 180,E1 1369.98,E2 1369.98} C_VEL
LIN {X 0,Y 592.938,Z 1077.46,A -85,B 0,C 180,E1 1373.478,E2 1373.478} C_VEL
LIN {X 0,Y 593.494,Z 1044.01,A -85,B 0,C 180,E1 1376.589,E2 1376.589} C_VEL
LIN {X 0,Y 594.149,Z 1007.418,A -85,B 0,C 180,E1 1379.227,E2 1379.227} C_VEL
LIN {X 0,Y 594.748,Z 968.127,A -85,B 0,C 180,E1 1381.359,E2 1381.359} C_VEL
LIN {X 0,Y 595.316,Z 926.802,A -85,B 0,C 180,E1 1382.921,E2 1382.921} C_VEL
LIN {X 0,Y 595.543,Z 888.407,A -85,B 0,C 180,E1 1383.812,E2 1383.812} C_VEL
LIN {X 0,Y 594.767,Z 851.023,A -85,B 0,C 180,E1 1384.416,E2 1384.416} C_VEL
LIN {X 0,Y 591.656,Z 843.44,A -85,B 0,C 180,E1 1384.811,E2 1384.811} C_VEL
LIN {X 0,Y 591.514,Z 843.44,A -85,B 0,C 180,E1 1390.066,E2 1390.066} C_VEL
LIN {X 0,Y 591.597,Z 843.44,A -85,B 0,C 180,E1 1395.579,E2 1395.579} C_VEL
LIN {X 0,Y 591.561,Z 843.44,A -85,B 0,C 180,E1 1400.379,E2 1400.379} C_VEL
LIN {X 0,Y 591.458,Z 843.44,A -85,B 0,C 180,E1 1405.856,E2 1405.856} C_VEL
LIN {X 0,Y 591.576,Z 843.44,A -85,B 0,C 180,E1 1411.011,E2 1411.011} C_VEL
LIN {X 0,Y 591.664,Z 843.44,A -85,B 0,C 180,E1 1415.917,E2 1415.917} C_VEL
LIN {X 0,Y 591.845,Z 843.44,A -85,B 0,C 180,E1 1420.643,E2 1420.643} C_VEL
LIN {X 0,Y 591.543,Z 843.44,A -85,B 0,C 180,E1 1425.221,E2 1425.221} C_VEL
LIN {X 0,Y 591.88,Z 843.44,A -85,B 0,C 180,E1 1429.72,E2 1429.72} C_VEL
LIN {X 0,Y 592.084,Z 843.44,A -85,B 0,C 180,E1 1434.149,E2 1434.149} C_VEL
LIN {X 0,Y 591.789,Z 843.44,A -85,B 0,C 180,E1 1440,E2 1440} C_VEL
LIN {X 0,Y 591.837,Z 843.44,A -85,B 0,C 180,E1 1444.387,E2 1444.387} C_VEL
LIN {X 0,Y 591.907,Z 843.44,A -85,B 0,C 180,E1 1448.798,E2 1448.798} C_VEL
LIN {X 0,Y 591.672,Z 843.44,A -85,B 0,C 180,E1 1454.266,E2 1454.266} C_VEL
LIN {X 0,Y 591.706,Z 843.44,A -85,B 0,C 180,E1 1459.361,E2 1459.361} C_VEL
LIN {X 0,Y 591.622,Z 843.44,A -85,B 0,C 180,E1 1464.084,E2 1464.084} C_VEL
LIN {X 0,Y 591.659,Z 843.44,A -85,B 0,C 180,E1 1468.984,E2 1468.984} C_VEL
LIN {X 0,Y 591.909,Z 843.44,A -85,B 0,C 180,E1 1474.114,E2 1474.114} C_VEL
LIN {X 0,Y 591.557,Z 843.44,A -85,B 0,C 180,E1 1480.068,E2 1480.068} C_VEL
LIN {X 0,Y 591.384,Z 843.44,A -85,B 0,C 180,E1 1485.597,E2 1485.597} C_VEL
LIN {X 0,Y 591.537,Z 843.44,A -85,B 0,C 180,E1 1490.375,E2 1490.375} C_VEL
LIN {X 0,Y 591.821,Z 843.44,A -85,B 0,C 180,E1 1495.659,E2 1495.659} C_VEL
LIN {X 0,Y 595.16,Z 852.426,A -85,B 0,C 180,E1 1496.017,E2 1496.017} C_VEL
LIN {X 0,Y 595.205,Z 897.094,A -85,B 0,C 180,E1 1497.037,E2 1497.037} C_VEL
LIN {X 0,Y 594.794,Z 937.872,A -85,B 0,C 180,E1 1498.587,E2 1498.587} C_VEL
LIN {X 0,Y 594.168,Z 976.813,A -85,B 0,C 180,E1 1500.691,E2 1500.691} C_VEL
LIN {X 0,Y 593.53,Z 1013.421,A -85,B 0,C 180,E1 1503.32,E2 1503.32} C_VEL
LIN {X 0,Y 592.917,Z 1046.477,A -85,B 0,C 180,E1 1506.375,E2 1506.375} C_VEL
LIN {X 0,Y 592.478,Z 1074.527,A -85,B 0,C 180,E1 1509.667,E2 1509.667} C_VEL
LIN {X 0,Y 592.16,Z 1098.392,A -85,B 0,C 180,E1 1513.239,E2 1513.239} C_VEL
LIN {X 0,Y 592.047,Z 1116.41,A -85,B 0,C 180,E1 1516.739,E2 1516.739} C_VEL
LIN {X 0,Y 591.915,Z 1130.375,A -85,B 0,C 180,E1 1520.461,E2 1520.461} C_VEL
LIN {X 0,Y 591.862,Z 1139.599,A -85,B 0,C 180,E1 1524.146,E2 1524.146} C_VEL
LIN {X 0,Y 592.03,Z 1143.678,A -85,B 0,C 180,E1 1527.078,E2 1527.078} C_VEL
LIN {X 0,Y 592.08,Z 1144.633,A -85,B 0,C 180,E1 1531.46,E2 1531.46} C_VEL
LIN {X 0,Y 592.023,Z 1139.427,A -85,B 0,C 180,E1 1535.852,E2 1535.852} C_VEL
LIN {X 0,Y 591.953,Z 1128.946,A -85,B 0,C 180,E1 1539.908,E2 1539.908} C_VEL
LIN {X 0,Y 592.045,Z 1113.272,A -85,B 0,C 180,E1 1543.845,E2 1543.845} C_VEL
LIN {X 0,Y 592.241,Z 1093.176,A -85,B 0,C 180,E1 1547.534,E2 1547.534} C_VEL
LIN {X 0,Y 592.672,Z 1067.929,A -85,B 0,C 180,E1 1551.091,E2 1551.091} C_VEL
LIN {X 0,Y 593.13,Z 1038.186,A -85,B 0,C 180,E1 1554.375,E2 1554.375} C_VEL
LIN {X 0,Y 593.732,Z 1003.012,A -85,B 0,C 180,E1 1557.411,E2 1557.411} C_VEL
LIN {X 0,Y 594.357,Z 965.209,A -85,B 0,C 180,E1 1559.917,E2 1559.917} C_VEL
LIN {X 0,Y 594.986,Z 925.62,A -85,B 0,C 180,E1 1561.855,E2 1561.855} C_VEL
LIN {X 0,Y 595.397,Z 886.481,A -85,B 0,C 180,E1 1563.162,E2 1563.162} C_VEL
LIN {X 0,Y 594.591,Z 850.41,A -85,B 0,C 180,E1 1563.962,E2 1563.962} C_VEL
LIN {X 0,Y 591.76,Z 843.44,A -85,B 0,C 180,E1 1564.331,E2 1564.331} C_VEL
LIN {X 0,Y 591.474,Z 843.44,A -85,B 0,C 180,E1 1570.062,E2 1570.062} C_VEL
LIN {X 0,Y 591.588,Z 843.44,A -85,B 0,C 180,E1 1575.579,E2 1575.579} C_VEL
LIN {X 0,Y 591.549,Z 843.44,A -85,B 0,C 180,E1 1580.379,E2 1580.379} C_VEL
LIN {X 0,Y 591.448,Z 843.44,A -85,B 0,C 180,E1 1585.856,E2 1585.856} C_VEL
LIN {X 0,Y 591.568,Z 843.44,A -85,B 0,C 180,E1 1591.011,E2 1591.011} C_VEL
LIN {X 0,Y 591.646,Z 843.44,A -85,B 0,C 180,E1 1595.917,E2 1595.917} C_VEL
LIN {X 0,Y 591.892,Z 843.44,A -85,B 0,C 180,E1 1600.645,E2 1600.645} C_VEL
LIN {X 0,Y 592.015,Z 843.44,A -85,B 0,C 180,E1 1606.739,E2 1606.739} C_VEL
LIN {X 0,Y 591.835,Z 843.44,A -85,B 0,C 180,E1 1612.711,E2 1612.711} C_VEL
LIN {X 0,Y 591.926,Z 843.44,A -85,B 0,C 180,E1 1617.078,E2 1617.078} C_VEL
LIN {X 0,Y 591.792,Z 843.44,A -85,B 0,C 180,E1 1622.451,E2 1622.451} C_VEL
LIN {X 0,Y 587.75,Z 843.44,A -85,B 0,C 180,E1 1624.108,E2 1624.108} C_VEL
LIN {X 0,Y 584.102,Z 843.44,A -85,B 0,C 180,E1 1625.787,E2 1625.787} C_VEL
LIN {X 0,Y 583.805,Z 843.44,A -85,B 0,C 180,E1 1631.934,E2 1631.934} C_VEL
LIN {X 0,Y 583.734,Z 843.44,A -85,B 0,C 180,E1 1636.964,E2 1636.964} C_VEL
LIN {X 0,Y 583.753,Z 843.44,A -85,B 0,C 180,E1 1641.471,E2 1641.471} C_VEL
LIN {X 0,Y 583.82,Z 843.44,A -85,B 0,C 180,E1 1646.065,E2 1646.065} C_VEL
LIN {X 0,Y 583.599,Z 843.44,A -85,B 0,C 180,E1 1651.43,E2 1651.43} C_VEL
LIN {X 0,Y 583.734,Z 843.44,A -85,B 0,C 180,E1 1656.738,E2 1656.738} C_VEL
LIN {X 0,Y 583.734,Z 843.44,A -85,B 0,C 180,E1 1662.23,E2 1662.23} C_VEL
LIN {X 0,Y 583.525,Z 843.44,A -85,B 0,C 180,E1 1667.75,E2 1667.75} C_VEL
LIN {X 0,Y 583.499,Z 843.44,A -85,B 0,C 180,E1 1673.29,E2 1673.29} C_VEL
LIN {X 0,Y 583.644,Z 843.44,A -85,B 0,C 180,E1 1674.705,E2 1674.705} C_VEL
LIN {X 0,Y 588.877,Z 856.49,A -85,B 0,C 180,E1 1675.27,E2 1675.27} C_VEL
LIN {X 0,Y 588.757,Z 910.753,A -85,B 0,C 180,E1 1676.209,E2 1676.209} C_VEL
LIN {X 0,Y 588.1,Z 954.388,A -85,B 0,C 180,E1 1677.63,E2 1677.63} C_VEL
LIN {X 0,Y 587.261,Z 997.219,A -85,B 0,C 180,E1 1679.754,E2 1679.754} C_VEL
LIN {X 0,Y 586.402,Z 1036.068,A -85,B 0,C 180,E1 1682.406,E2 1682.406} C_VEL
LIN {X 0,Y 585.6,Z 1070.624,A -85,B 0,C 180,E1 1685.488,E2 1685.488} C_VEL
LIN {X 0,Y 584.895,Z 1101.46,A -85,B 0,C 180,E1 1689.024,E2 1689.024} C_VEL
LIN {X 0,Y 584.42,Z 1127.002,A -85,B 0,C 180,E1 1692.81,E2 1692.81} C_VEL
LIN {X 0,Y 584.221,Z 1146.203,A -85,B 0,C 180,E1 1696.558,E2 1696.558} C_VEL
LIN {X 0,Y 584.045,Z 1160.236,A -85,B 0,C 180,E1 1700.332,E2 1700.332} C_VEL
LIN {X 0,Y 584.01,Z 1169.517,A -85,B 0,C 180,E1 1704.068,E2 1704.068} C_VEL
LIN {X 0,Y 584.127,Z 1173.637,A -85,B 0,C 180,E1 1707.039,E2 1707.039} C_VEL
LIN {X 0,Y 584.232,Z 1174.659,A -85,B 0,C 180,E1 1711.48,E2 1711.48} C_VEL
LIN {X 0,Y 583.99,Z 1170.73,A -85,B 0,C 180,E1 1715.189,E2 1715.189} C_VEL
LIN {X 0,Y 584.01,Z 1162.53,A -85,B 0,C 180,E1 1718.919,E2 1718.919} C_VEL
LIN {X 0,Y 584.102,Z 1149.391,A -85,B 0,C 180,E1 1722.685,E2 1722.685} C_VEL
LIN {X 0,Y 584.397,Z 1130.909,A -85,B 0,C 180,E1 1726.502,E2 1726.502} C_VEL
LIN {X 0,Y 584.801,Z 1106.899,A -85,B 0,C 180,E1 1730.248,E2 1730.248} C_VEL
LIN {X 0,Y 585.4,Z 1077.459,A -85,B 0,C 180,E1 1733.798,E2 1733.798} C_VEL
LIN {X 0,Y 586.201,Z 1044.444,A -85,B 0,C 180,E1 1736.91,E2 1736.91} C_VEL
LIN {X 0,Y 587.028,Z 1008.388,A -85,B 0,C 180,E1 1739.556,E2 1739.556} C_VEL
LIN {X 0,Y 587.84,Z 969.67,A -85,B 0,C 180,E1 1741.699,E2 1741.699} C_VEL
LIN {X 0,Y 588.582,Z 928.242,A -85,B 0,C 180,E1 1743.298,E2 1743.298} C_VEL
LIN {X 0,Y 588.978,Z 890.469,A -85,B 0,C 180,E1 1744.206,E2 1744.206} C_VEL
LIN {X 0,Y 588.181,Z 853.544,A -85,B 0,C 180,E1 1744.82,E2 1744.82} C_VEL
LIN {X 0,Y 583.641,Z 843.44,A -85,B 0,C 180,E1 1745.296,E2 1745.296} C_VEL
LIN {X 0,Y 583.534,Z 843.44,A -85,B 0,C 180,E1 1751.417,E2 1751.417} C_VEL
LIN {X 0,Y 583.72,Z 843.44,A -85,B 0,C 180,E1 1756.373,E2 1756.373} C_VEL
LIN {X 0,Y 583.678,Z 843.44,A -85,B 0,C 180,E1 1761.65,E2 1761.65} C_VEL
LIN {X 0,Y 583.518,Z 843.44,A -85,B 0,C 180,E1 1767.108,E2 1767.108} C_VEL
LIN {X 0,Y 583.606,Z 843.44,A -85,B 0,C 180,E1 1772.264,E2 1772.264} C_VEL
LIN {X 0,Y 583.62,Z 843.44,A -85,B 0,C 180,E1 1777.181,E2 1777.181} C_VEL
LIN {X 0,Y 583.893,Z 843.44,A -85,B 0,C 180,E1 1781.934,E2 1781.934} C_VEL
LIN {X 0,Y 583.698,Z 843.44,A -85,B 0,C 180,E1 1788.064,E2 1788.064} C_VEL
LIN {X 0,Y 584.164,Z 843.44,A -85,B 0,C 180,E1 1794.069,E2 1794.069} C_VEL
LIN {X 0,Y 583.911,Z 843.44,A -85,B 0,C 180,E1 1800,E2 1800} C_VEL
LIN {X 0,Y 583.94,Z 843.44,A -85,B 0,C 180,E1 1804.446,E2 1804.446} C_VEL
LIN {X 0,Y 583.968,Z 843.44,A -85,B 0,C 180,E1 1808.919,E2 1808.919} C_VEL
LIN {X 0,Y 583.982,Z 843.44,A -85,B 0,C 180,E1 1813.447,E2 1813.447} C_VEL
LIN {X 0,Y 583.933,Z 843.44,A -85,B 0,C 180,E1 1818.065,E2 1818.065} C_VEL
LIN {X 0,Y 583.825,Z 843.44,A -85,B 0,C 180,E1 1822.811,E2 1822.811} C_VEL
LIN {X 0,Y 583.723,Z 843.44,A -85,B 0,C 180,E1 1828.483,E2 1828.483} C_VEL
LIN {X 0,Y 583.921,Z 843.44,A -85,B 0,C 180,E1 1834.647,E2 1834.647} C_VEL
LIN {X 0,Y 583.637,Z 843.44,A -85,B 0,C 180,E1 1840.267,E2 1840.267} C_VEL
LIN {X 0,Y 583.58,Z 843.44,A -85,B 0,C 180,E1 1846.385,E2 1846.385} C_VEL
LIN {X 0,Y 583.698,Z 843.44,A -85,B 0,C 180,E1 1851.65,E2 1851.65} C_VEL
LIN {X 0,Y 583.862,Z 843.44,A -85,B 0,C 180,E1 1855.124,E2 1855.124} C_VEL
LIN {X 0,Y 588.639,Z 855.279,A -85,B 0,C 180,E1 1855.638,E2 1855.638} C_VEL
LIN {X 0,Y 588.495,Z 897.98,A -85,B 0,C 180,E1 1856.643,E2 1856.643} C_VEL
LIN {X 0,Y 587.907,Z 939.069,A -85,B 0,C 180,E1 1858.231,E2 1858.231} C_VEL
LIN {X 0,Y 587.026,Z 979.184,A -85,B 0,C 180,E1 1860.449,E2 1860.449} C_VEL
LIN {X 0,Y 586.097,Z 1018.126,A -85,B 0,C 180,E1 1863.348,E2 1863.348} C_VEL
LIN {X 0,Y 585.323,Z 1051.557,A -85,B 0,C 180,E1 1866.596,E2 1866.596} C_VEL
LIN {X 0,Y 584.71,Z 1080.423,A -85,B 0,C 180,E1 1870.196,E2 1870.196} C_VEL
LIN {X 0,Y 584.331,Z 1103.34,A -85,B 0,C 180,E1 1873.882,E2 1873.882} C_VEL
LIN {X 0,Y 584.151,Z 1121.118,A -85,B 0,C 180,E1 1877.695,E2 1877.695} C_VEL
LIN {X 0,Y 583.994,Z 1132.659,A -85,B 0,C 180,E1 1881.081,E2 1881.081} C_VEL
LIN {X 0,Y 583.942,Z 1140.803,A -85,B 0,C 180,E1 1884.811,E2 1884.811} C_VEL
LIN {X 0,Y 583.973,Z 1144.678,A -85,B 0,C 180,E1 1888.519,E2 1888.519} C_VEL
LIN {X 0,Y 584.19,Z 1144.633,A -85,B 0,C 180,E1 1891.48,E2 1891.48} C_VEL
LIN {X 0,Y 584.122,Z 1139.428,A -85,B 0,C 180,E1 1895.931,E2 1895.931} C_VEL
LIN {X 0,Y 584.062,Z 1128.948,A -85,B 0,C 180,E1 1900.043,E2 1900.043} C_VEL
LIN {X 0,Y 584.216,Z 1113.572,A -85,B 0,C 180,E1 1903.97,E2 1903.97} C_VEL
LIN {X 0,Y 584.454,Z 1094.437,A -85,B 0,C 180,E1 1907.574,E2 1907.574} C_VEL
LIN {X 0,Y 584.996,Z 1068.395,A -85,B 0,C 180,E1 1911.324,E2 1911.324} C_VEL
LIN {X 0,Y 585.635,Z 1038.543,A -85,B 0,C 180,E1 1914.674,E2 1914.674} C_VEL
LIN {X 0,Y 586.472,Z 1003.091,A -85,B 0,C 180,E1 1917.774,E2 1917.774} C_VEL
LIN {X 0,Y 587.349,Z 964.607,A -85,B 0,C 180,E1 1920.347,E2 1920.347} C_VEL
LIN {X 0,Y 588.195,Z 925.349,A -85,B 0,C 180,E1 1922.279,E2 1922.279} C_VEL
LIN {X 0,Y 588.746,Z 886.509,A -85,B 0,C 180,E1 1923.586,E2 1923.586} C_VEL
LIN {X 0,Y 588.11,Z 853.26,A -85,B 0,C 180,E1 1924.342,E2 1924.342} C_VEL
LIN {X 0,Y 583.721,Z 843.44,A -85,B 0,C 180,E1 1924.849,E2 1924.849} C_VEL
LIN {X 0,Y 583.541,Z 843.44,A -85,B 0,C 180,E1 1930.277,E2 1930.277} C_VEL
LIN {X 0,Y 583.695,Z 843.44,A -85,B 0,C 180,E1 1935.734,E2 1935.734} C_VEL
LIN {X 0,Y 583.671,Z 843.44,A -85,B 0,C 180,E1 1941.65,E2 1941.65} C_VEL
LIN {X 0,Y 583.51,Z 843.44,A -85,B 0,C 180,E1 1947.108,E2 1947.108} C_VEL
LIN {X 0,Y 583.597,Z 843.44,A -85,B 0,C 180,E1 1952.263,E2 1952.263} C_VEL
LIN {X 0,Y 583.623,Z 843.44,A -85,B 0,C 180,E1 1957.181,E2 1957.181} C_VEL
LIN {X 0,Y 583.886,Z 843.44,A -85,B 0,C 180,E1 1961.934,E2 1961.934} C_VEL
LIN {X 0,Y 584.1,Z 843.44,A -85,B 0,C 180,E1 1966.556,E2 1966.556} C_VEL
LIN {X 0,Y 583.911,Z 843.44,A -85,B 0,C 180,E1 1972.696,E2 1972.696} C_VEL
LIN {X 0,Y 584.042,Z 843.44,A -85,B 0,C 180,E1 1977.038,E2 1977.038} C_VEL
LIN {X 0,Y 583.909,Z 843.44,A -85,B 0,C 180,E1 1982.437,E2 1982.437} C_VEL
LIN {X 0,Y 584.102,Z 843.44,A -85,B 0,C 180,E1 1985.787,E2 1985.787} C_VEL
LIN {X 0,Y 581.641,Z 843.44,A -85,B 0,C 180,E1 1987.048,E2 1987.048} C_VEL
LIN {X 0,Y 575.989,Z 843.44,A -85,B 0,C 180,E1 1988.933,E2 1988.933} C_VEL
LIN {X 0,Y 575.888,Z 843.44,A -85,B 0,C 180,E1 1989.151,E2 1989.151} C_VEL
LIN {X 0,Y 575.933,Z 843.44,A -85,B 0,C 180,E1 1995.189,E2 1995.189} C_VEL
LIN {X 0,Y 575.859,Z 843.44,A -85,B 0,C 180,E1 2001.522,E2 2001.522} C_VEL
LIN {X 0,Y 575.791,Z 843.44,A -85,B 0,C 180,E1 2006.993,E2 2006.993} C_VEL
LIN {X 0,Y 575.688,Z 843.44,A -85,B 0,C 180,E1 2011.616,E2 2011.616} C_VEL
LIN {X 0,Y 575.817,Z 843.44,A -85,B 0,C 180,E1 2017.065,E2 2017.065} C_VEL
LIN {X 0,Y 575.797,Z 843.44,A -85,B 0,C 180,E1 2022.951,E2 2022.951} C_VEL
LIN {X 0,Y 575.63,Z 843.44,A -85,B 0,C 180,E1 2029.052,E2 2029.052} C_VEL
LIN {X 0,Y 575.669,Z 843.61,A -85,B 0,C 180,E1 2034.159,E2 2034.159} C_VEL
LIN {X 0,Y 582.388,Z 859.124,A -85,B 0,C 180,E1 2034.865,E2 2034.865} C_VEL
LIN {X 0,Y 582.15,Z 911.386,A -85,B 0,C 180,E1 2035.79,E2 2035.79} C_VEL
LIN {X 0,Y 581.3,Z 954.517,A -85,B 0,C 180,E1 2037.209,E2 2037.209} C_VEL
LIN {X 0,Y 580.221,Z 997.237,A -85,B 0,C 180,E1 2039.349,E2 2039.349} C_VEL
LIN {X 0,Y 579.118,Z 1036.065,A -85,B 0,C 180,E1 2042.029,E2 2042.029} C_VEL
LIN {X 0,Y 578.095,Z 1070.832,A -85,B 0,C 180,E1 2045.17,E2 2045.17} C_VEL
LIN {X 0,Y 577.25,Z 1101.462,A -85,B 0,C 180,E1 2048.733,E2 2048.733} C_VEL
LIN {X 0,Y 576.662,Z 1127.004,A -85,B 0,C 180,E1 2052.571,E2 2052.571} C_VEL
LIN {X 0,Y 576.397,Z 1146.202,A -85,B 0,C 180,E1 2056.372,E2 2056.372} C_VEL
LIN {X 0,Y 576.193,Z 1160.237,A -85,B 0,C 180,E1 2060.199,E2 2060.199} C_VEL
LIN {X 0,Y 576.131,Z 1169.517,A -85,B 0,C 180,E1 2063.986,E2 2063.986} C_VEL
LIN {X 0,Y 576.216,Z 1173.637,A -85,B 0,C 180,E1 2066.998,E2 2066.998} C_VEL
LIN {X 0,Y 576.328,Z 1174.659,A -85,B 0,C 180,E1 2071.501,E2 2071.501} C_VEL
LIN {X 0,Y 576.132,Z 1169.517,A -85,B 0,C 180,E1 2076.014,E2 2076.014} C_VEL
LIN {X 0,Y 576.199,Z 1159.086,A -85,B 0,C 180,E1 2080.182,E2 2080.182} C_VEL
LIN {X 0,Y 576.33,Z 1144.462,A -85,B 0,C 180,E1 2084.015,E2 2084.015} C_VEL
LIN {X 0,Y 576.729,Z 1124.453,A -85,B 0,C 180,E1 2087.86,E2 2087.86} C_VEL
LIN {X 0,Y 577.302,Z 1098.747,A -85,B 0,C 180,E1 2091.623,E2 2091.623} C_VEL
LIN {X 0,Y 578.145,Z 1068.03,A -85,B 0,C 180,E1 2095.112,E2 2095.112} C_VEL
LIN {X 0,Y 579.194,Z 1033.049,A -85,B 0,C 180,E1 2098.203,E2 2098.203} C_VEL
LIN {X 0,Y 580.33,Z 995.368,A -85,B 0,C 180,E1 2100.755,E2 2100.755} C_VEL
LIN {X 0,Y 581.4,Z 954.427,A -85,B 0,C 180,E1 2102.788,E2 2102.788} C_VEL
LIN {X 0,Y 582.112,Z 911.167,A -85,B 0,C 180,E1 2104.219,E2 2104.219} C_VEL
LIN {X 0,Y 581.753,Z 856.826,A -85,B 0,C 180,E1 2105.213,E2 2105.213} C_VEL
LIN {X 0,Y 575.806,Z 844.819,A -85,B 0,C 180,E1 2105.812,E2 2105.812} C_VEL
LIN {X 0,Y 575.675,Z 843.44,A -85,B 0,C 180,E1 2105.877,E2 2105.877} C_VEL
LIN {X 0,Y 575.635,Z 843.44,A -85,B 0,C 180,E1 2110.948,E2 2110.948} C_VEL
LIN {X 0,Y 575.79,Z 843.44,A -85,B 0,C 180,E1 2117.208,E2 2117.208} C_VEL
LIN {X 0,Y 575.809,Z 843.44,A -85,B 0,C 180,E1 2122.934,E2 2122.934} C_VEL
LIN {X 0,Y 575.735,Z 843.44,A -85,B 0,C 180,E1 2128.387,E2 2128.387} C_VEL
LIN {X 0,Y 575.818,Z 843.44,A -85,B 0,C 180,E1 2133.545,E2 2133.545} C_VEL
LIN {X 0,Y 575.972,Z 843.44,A -85,B 0,C 180,E1 2140.088,E2 2140.088} C_VEL
LIN {X 0,Y 575.801,Z 843.44,A -85,B 0,C 180,E1 2144.807,E2 2144.807} C_VEL
LIN {X 0,Y 575.895,Z 843.44,A -85,B 0,C 180,E1 2150.955,E2 2150.955} C_VEL
LIN {X 0,Y 575.967,Z 843.44,A -85,B 0,C 180,E1 2155.492,E2 2155.492} C_VEL
LIN {X 0,Y 576.01,Z 843.44,A -85,B 0,C 180,E1 2160,E2 2160} C_VEL
LIN {X 0,Y 575.916,Z 843.44,A -85,B 0,C 180,E1 2165.329,E2 2165.329} C_VEL
LIN {X 0,Y 575.838,Z 843.44,A -85,B 0,C 180,E1 2170.57,E2 2170.57} C_VEL
LIN {X 0,Y 575.812,Z 843.44,A -85,B 0,C 180,E1 2175.192,E2 2175.192} C_VEL
LIN {X 0,Y 575.853,Z 843.44,A -85,B 0,C 180,E1 2179.916,E2 2179.916} C_VEL
LIN {X 0,Y 575.73,Z 843.44,A -85,B 0,C 180,E1 2184.793,E2 2184.793} C_VEL
LIN {X 0,Y 575.727,Z 843.44,A -85,B 0,C 180,E1 2190.123,E2 2190.123} C_VEL
LIN {X 0,Y 575.919,Z 843.44,A -85,B 0,C 180,E1 2195.199,E2 2195.199} C_VEL
LIN {X 0,Y 575.723,Z 843.44,A -85,B 0,C 180,E1 2200.938,E2 2200.938} C_VEL
LIN {X 0,Y 575.748,Z 843.44,A -85,B 0,C 180,E1 2207.209,E2 2207.209} C_VEL
LIN {X 0,Y 575.836,Z 843.44,A -85,B 0,C 180,E1 2212.934,E2 2212.934} C_VEL
LIN {X 0,Y 575.929,Z 843.45,A -85,B 0,C 180,E1 2214.581,E2 2214.581} C_VEL
LIN {X 0,Y 582.157,Z 859.069,A -85,B 0,C 180,E1 2215.267,E2 2215.267} C_VEL
LIN {X 0,Y 581.782,Z 900.549,A -85,B 0,C 180,E1 2216.295,E2 2216.295} C_VEL
LIN {X 0,Y 581.038,Z 939.759,A -85,B 0,C 180,E1 2217.846,E2 2217.846} C_VEL
LIN {X 0,Y 579.897,Z 980.413,A -85,B 0,C 180,E1 2220.13,E2 2220.13} C_VEL
LIN {X 0,Y 578.759,Z 1018.754,A -85,B 0,C 180,E1 2223.041,E2 2223.041} C_VEL
LIN {X 0,Y 577.747,Z 1052.337,A -85,B 0,C 180,E1 2226.362,E2 2226.362} C_VEL
LIN {X 0,Y 577.032,Z 1080.448,A -85,B 0,C 180,E1 2229.926,E2 2229.926} C_VEL
LIN {X 0,Y 576.544,Z 1103.335,A -85,B 0,C 180,E1 2233.658,E2 2233.658} C_VEL
LIN {X 0,Y 576.298,Z 1121.116,A -85,B 0,C 180,E1 2237.524,E2 2237.524} C_VEL
LIN {X 0,Y 576.11,Z 1132.657,A -85,B 0,C 180,E1 2240.958,E2 2240.958} C_VEL
LIN {X 0,Y 576.08,Z 1140.374,A -85,B 0,C 180,E1 2244.471,E2 2244.471} C_VEL
LIN {X 0,Y 576.073,Z 1144.678,A -85,B 0,C 180,E1 2248.499,E2 2248.499} C_VEL
LIN {X 0,Y 576.284,Z 1144.634,A -85,B 0,C 180,E1 2251.5,E2 2251.5} C_VEL
LIN {X 0,Y 576.218,Z 1139.43,A -85,B 0,C 180,E1 2256.013,E2 2256.013} C_VEL
LIN {X 0,Y 576.165,Z 1128.95,A -85,B 0,C 180,E1 2260.183,E2 2260.183} C_VEL
LIN {X 0,Y 576.358,Z 1114.281,A -85,B 0,C 180,E1 2264.009,E2 2264.009} C_VEL
LIN {X 0,Y 576.718,Z 1094.077,A -85,B 0,C 180,E1 2267.878,E2 2267.878} C_VEL
LIN {X 0,Y 577.324,Z 1068.399,A -85,B 0,C 180,E1 2271.622,E2 2271.622} C_VEL
LIN {X 0,Y 578.183,Z 1037.558,A -85,B 0,C 180,E1 2275.112,E2 2275.112} C_VEL
LIN {X 0,Y 579.236,Z 1002.424,A -85,B 0,C 180,E1 2278.204,E2 2278.204} C_VEL
LIN {X 0,Y 580.354,Z 964.489,A -85,B 0,C 180,E1 2280.759,E2 2280.759} C_VEL
LIN {X 0,Y 581.427,Z 924.546,A -85,B 0,C 180,E1 2282.736,E2 2282.736} C_VEL
LIN {X 0,Y 582.161,Z 886.521,A -85,B 0,C 180,E1 2284.018,E2 2284.018} C_VEL
LIN {X 0,Y 581.713,Z 856.649,A -85,B 0,C 180,E1 2284.715,E2 2284.715} C_VEL
LIN {X 0,Y 575.715,Z 843.44,A -85,B 0,C 180,E1 2285.387,E2 2285.387} C_VEL
LIN {X 0,Y 575.605,Z 843.44,A -85,B 0,C 180,E1 2290.95,E2 2290.95} C_VEL
LIN {X 0,Y 575.787,Z 843.44,A -85,B 0,C 180,E1 2297.049,E2 2297.049} C_VEL
LIN {X 0,Y 575.797,Z 843.44,A -85,B 0,C 180,E1 2302.933,E2 2302.933} C_VEL
LIN {X 0,Y 575.727,Z 843.44,A -85,B 0,C 180,E1 2308.386,E2 2308.386} C_VEL
LIN {X 0,Y 575.8,Z 843.44,A -85,B 0,C 180,E1 2313.544,E2 2313.544} C_VEL
LIN {X 0,Y 576.035,Z 843.44,A -85,B 0,C 180,E1 2320.09,E2 2320.09} C_VEL
LIN {X 0,Y 576.154,Z 843.44,A -85,B 0,C 180,E1 2326.367,E2 2326.367} C_VEL
LIN {X 0,Y 575.987,Z 843.44,A -85,B 0,C 180,E1 2332.683,E2 2332.683} C_VEL
LIN {X 0,Y 576.134,Z 843.44,A -85,B 0,C 180,E1 2336.998,E2 2336.998} C_VEL
LIN {X 0,Y 576.256,Z 843.44,A -85,B 0,C 180,E1 2341.501,E2 2341.501} C_VEL
LIN {X 0,Y 576.233,Z 843.44,A -85,B 0,C 180,E1 2346.013,E2 2346.013} C_VEL
LIN {X 0,Y 575.888,Z 843.44,A -85,B 0,C 180,E1 2349.151,E2 2349.151} C_VEL
LIN {X 0,Y 574.644,Z 843.44,A -85,B 0,C 180,E1 2350.012,E2 2350.012} C_VEL
LIN {X 0,Y 568.034,Z 843.44,A -85,B 0,C 180,E1 2352.352,E2 2352.352} C_VEL
LIN {X 0,Y 567.922,Z 843.44,A -85,B 0,C 180,E1 2352.574,E2 2352.574} C_VEL
LIN {X 0,Y 567.95,Z 843.44,A -85,B 0,C 180,E1 2356.993,E2 2356.993} C_VEL
LIN {X 0,Y 567.904,Z 843.44,A -85,B 0,C 180,E1 2361.838,E2 2361.838} C_VEL
LIN {X 0,Y 567.898,Z 843.44,A -85,B 0,C 180,E1 2366.853,E2 2366.853} C_VEL
LIN {X 0,Y 567.74,Z 843.44,A -85,B 0,C 180,E1 2372.111,E2 2372.111} C_VEL
LIN {X 0,Y 567.889,Z 843.44,A -85,B 0,C 180,E1 2377.672,E2 2377.672} C_VEL
LIN {X 0,Y 567.796,Z 843.44,A -85,B 0,C 180,E1 2383.707,E2 2383.707} C_VEL
LIN {X 0,Y 567.664,Z 843.44,A -85,B 0,C 180,E1 2388.351,E2 2388.351} C_VEL
LIN {X 0,Y 567.727,Z 843.563,A -85,B 0,C 180,E1 2393.578,E2 2393.578} C_VEL
LIN {X 0,Y 575.912,Z 860.809,A -85,B 0,C 180,E1 2394.436,E2 2394.436} C_VEL
LIN {X 0,Y 575.575,Z 911.999,A -85,B 0,C 180,E1 2395.362,E2 2395.362} C_VEL
LIN {X 0,Y 574.566,Z 954.525,A -85,B 0,C 180,E1 2396.776,E2 2396.776} C_VEL
LIN {X 0,Y 573.252,Z 997.234,A -85,B 0,C 180,E1 2398.935,E2 2398.935} C_VEL
LIN {X 0,Y 571.897,Z 1036.062,A -85,B 0,C 180,E1 2401.644,E2 2401.644} C_VEL
LIN {X 0,Y 570.674,Z 1071.01,A -85,B 0,C 180,E1 2404.845,E2 2404.845} C_VEL
LIN {X 0,Y 569.605,Z 1101.464,A -85,B 0,C 180,E1 2408.434,E2 2408.434} C_VEL
LIN {X 0,Y 568.973,Z 1126.099,A -85,B 0,C 180,E1 2412.164,E2 2412.164} C_VEL
LIN {X 0,Y 568.593,Z 1146.201,A -85,B 0,C 180,E1 2416.181,E2 2416.181} C_VEL
LIN {X 0,Y 568.285,Z 1161.388,A -85,B 0,C 180,E1 2420.447,E2 2420.447} C_VEL
LIN {X 0,Y 568.194,Z 1170.354,A -85,B 0,C 180,E1 2424.427,E2 2424.427} C_VEL
LIN {X 0,Y 568.17,Z 1174.659,A -85,B 0,C 180,E1 2428.478,E2 2428.478} C_VEL
LIN {X 0,Y 568.444,Z 1174.659,A -85,B 0,C 180,E1 2431.521,E2 2431.521} C_VEL
LIN {X 0,Y 568.24,Z 1169.517,A -85,B 0,C 180,E1 2436.098,E2 2436.098} C_VEL
LIN {X 0,Y 568.35,Z 1159.086,A -85,B 0,C 180,E1 2440.324,E2 2440.324} C_VEL
LIN {X 0,Y 568.516,Z 1144.463,A -85,B 0,C 180,E1 2444.211,E2 2444.211} C_VEL
LIN {X 0,Y 569.015,Z 1123.946,A -85,B 0,C 180,E1 2448.195,E2 2448.195} C_VEL
LIN {X 0,Y 569.687,Z 1098.033,A -85,B 0,C 180,E1 2452.019,E2 2452.019} C_VEL
LIN {X 0,Y 570.748,Z 1067.413,A -85,B 0,C 180,E1 2455.523,E2 2455.523} C_VEL
LIN {X 0,Y 571.967,Z 1034.163,A -85,B 0,C 180,E1 2458.505,E2 2458.505} C_VEL
LIN {X 0,Y 573.364,Z 995.765,A -85,B 0,C 180,E1 2461.147,E2 2461.147} C_VEL
LIN {X 0,Y 574.616,Z 954.437,A -85,B 0,C 180,E1 2463.224,E2 2463.224} C_VEL
LIN {X 0,Y 575.562,Z 911.022,A -85,B 0,C 180,E1 2464.667,E2 2464.667} C_VEL
LIN {X 0,Y 575.409,Z 859.824,A -85,B 0,C 180,E1 2465.615,E2 2465.615} C_VEL
LIN {X 0,Y 567.889,Z 845.067,A -85,B 0,C 180,E1 2466.387,E2 2466.387} C_VEL
LIN {X 0,Y 567.71,Z 843.44,A -85,B 0,C 180,E1 2466.476,E2 2466.476} C_VEL
LIN {X 0,Y 567.672,Z 843.44,A -85,B 0,C 180,E1 2471.903,E2 2471.903} C_VEL
LIN {X 0,Y 567.798,Z 843.44,A -85,B 0,C 180,E1 2478.086,E2 2478.086} C_VEL
LIN {X 0,Y 567.821,Z 843.44,A -85,B 0,C 180,E1 2484.222,E2 2484.222} C_VEL
LIN {X 0,Y 567.833,Z 843.44,A -85,B 0,C 180,E1 2489.675,E2 2489.675} C_VEL
LIN {X 0,Y 567.912,Z 843.44,A -85,B 0,C 180,E1 2494.841,E2 2494.841} C_VEL
LIN {X 0,Y 568.019,Z 843.44,A -85,B 0,C 180,E1 2499.797,E2 2499.797} C_VEL
LIN {X 0,Y 567.91,Z 843.44,A -85,B 0,C 180,E1 2504.591,E2 2504.591} C_VEL
LIN {X 0,Y 567.989,Z 843.44,A -85,B 0,C 180,E1 2510.828,E2 2510.828} C_VEL
LIN {X 0,Y 568.077,Z 843.44,A -85,B 0,C 180,E1 2515.429,E2 2515.429} C_VEL
LIN {X 0,Y 568.135,Z 843.44,A -85,B 0,C 180,E1 2520,E2 2520} C_VEL
LIN {X 0,Y 568.114,Z 843.44,A -85,B 0,C 180,E1 2524.57,E2 2524.57} C_VEL
LIN {X 0,Y 568.111,Z 843.44,A -85,B 0,C 180,E1 2529.17,E2 2529.17} C_VEL
LIN {X 0,Y 568.103,Z 843.44,A -85,B 0,C 180,E1 2533.83,E2 2533.83} C_VEL
LIN {X 0,Y 568.053,Z 843.44,A -85,B 0,C 180,E1 2538.588,E2 2538.588} C_VEL
LIN {X 0,Y 567.937,Z 843.44,A -85,B 0,C 180,E1 2543.486,E2 2543.486} C_VEL
LIN {X 0,Y 567.859,Z 843.44,A -85,B 0,C 180,E1 2548.725,E2 2548.725} C_VEL
LIN {X 0,Y 567.994,Z 843.44,A -85,B 0,C 180,E1 2554.554,E2 2554.554} C_VEL
LIN {X 0,Y 567.81,Z 843.44,A -85,B 0,C 180,E1 2559.628,E2 2559.628} C_VEL
LIN {X 0,Y 567.649,Z 843.44,A -85,B 0,C 180,E1 2565.867,E2 2565.867} C_VEL
LIN {X 0,Y 567.803,Z 843.44,A -85,B 0,C 180,E1 2570.415,E2 2570.415} C_VEL
LIN {X 0,Y 568.023,Z 843.94,A -85,B 0,C 180,E1 2574.021,E2 2574.021} C_VEL
LIN {X 0,Y 575.696,Z 862.043,A -85,B 0,C 180,E1 2574.874,E2 2574.874} C_VEL
LIN {X 0,Y 575.047,Z 904.709,A -85,B 0,C 180,E1 2575.991,E2 2575.991} C_VEL
LIN {X 0,Y 574.096,Z 943.159,A -85,B 0,C 180,E1 2577.588,E2 2577.588} C_VEL
LIN {X 0,Y 572.785,Z 981.976,A -85,B 0,C 180,E1 2579.833,E2 2579.833} C_VEL
LIN {X 0,Y 571.464,Z 1018.225,A -85,B 0,C 180,E1 2582.62,E2 2582.62} C_VEL
LIN {X 0,Y 570.232,Z 1051.134,A -85,B 0,C 180,E1 2585.89,E2 2585.89} C_VEL
LIN {X 0,Y 569.344,Z 1080.445,A -85,B 0,C 180,E1 2589.643,E2 2589.643} C_VEL
LIN {X 0,Y 568.722,Z 1104.346,A -85,B 0,C 180,E1 2593.625,E2 2593.625} C_VEL
LIN {X 0,Y 568.439,Z 1122.648,A -85,B 0,C 180,E1 2597.738,E2 2597.738} C_VEL
LIN {X 0,Y 568.268,Z 1134.586,A -85,B 0,C 180,E1 2601.602,E2 2601.602} C_VEL
LIN {X 0,Y 568.141,Z 1141.985,A -85,B 0,C 180,E1 2605.43,E2 2605.43} C_VEL
LIN {X 0,Y 568.186,Z 1144.678,A -85,B 0,C 180,E1 2608.478,E2 2608.478} C_VEL
LIN {X 0,Y 568.4,Z 1144.634,A -85,B 0,C 180,E1 2611.521,E2 2611.521} C_VEL
LIN {X 0,Y 568.336,Z 1140.362,A -85,B 0,C 180,E1 2615.521,E2 2615.521} C_VEL
LIN {X 0,Y 568.374,Z 1131.253,A -85,B 0,C 180,E1 2619.551,E2 2619.551} C_VEL
LIN {X 0,Y 568.543,Z 1116.002,A -85,B 0,C 180,E1 2623.82,E2 2623.82} C_VEL
LIN {X 0,Y 568.908,Z 1095.709,A -85,B 0,C 180,E1 2627.86,E2 2627.86} C_VEL
LIN {X 0,Y 569.659,Z 1069.643,A -85,B 0,C 180,E1 2631.768,E2 2631.768} C_VEL
LIN {X 0,Y 570.755,Z 1038.138,A -85,B 0,C 180,E1 2635.404,E2 2635.404} C_VEL
LIN {X 0,Y 572.024,Z 1003.562,A -85,B 0,C 180,E1 2638.504,E2 2638.504} C_VEL
LIN {X 0,Y 573.364,Z 965.921,A -85,B 0,C 180,E1 2641.093,E2 2641.093} C_VEL
LIN {X 0,Y 574.65,Z 926.048,A -85,B 0,C 180,E1 2643.105,E2 2643.105} C_VEL
LIN {X 0,Y 575.516,Z 889.052,A -85,B 0,C 180,E1 2644.393,E2 2644.393} C_VEL
LIN {X 0,Y 575.193,Z 859.309,A -85,B 0,C 180,E1 2645.12,E2 2645.12} C_VEL
LIN {X 0,Y 567.734,Z 843.44,A -85,B 0,C 180,E1 2645.935,E2 2645.935} C_VEL
LIN {X 0,Y 567.655,Z 843.44,A -85,B 0,C 180,E1 2651.901,E2 2651.901} C_VEL
LIN {X 0,Y 567.797,Z 843.44,A -85,B 0,C 180,E1 2658.086,E2 2658.086} C_VEL
LIN {X 0,Y 567.807,Z 843.44,A -85,B 0,C 180,E1 2664.222,E2 2664.222} C_VEL
LIN {X 0,Y 567.826,Z 843.44,A -85,B 0,C 180,E1 2669.675,E2 2669.675} C_VEL
LIN {X 0,Y 567.895,Z 843.44,A -85,B 0,C 180,E1 2674.841,E2 2674.841} C_VEL
LIN {X 0,Y 568.07,Z 843.44,A -85,B 0,C 180,E1 2679.799,E2 2679.799} C_VEL
LIN {X 0,Y 568.234,Z 843.44,A -85,B 0,C 180,E1 2686.173,E2 2686.173} C_VEL
LIN {X 0,Y 568.063,Z 843.44,A -85,B 0,C 180,E1 2692.671,E2 2692.671} C_VEL
LIN {X 0,Y 568.229,Z 843.44,A -85,B 0,C 180,E1 2696.956,E2 2696.956} C_VEL
LIN {X 0,Y 568.369,Z 843.44,A -85,B 0,C 180,E1 2701.521,E2 2701.521} C_VEL
LIN {X 0,Y 568.299,Z 843.44,A -85,B 0,C 180,E1 2706.097,E2 2706.097} C_VEL
LIN {X 0,Y 567.961,Z 843.44,A -85,B 0,C 180,E1 2712.272,E2 2712.272} C_VEL
LIN {X 0,Y 567.922,Z 843.44,A -85,B 0,C 180,E1 2712.574,E2 2712.574} C_VEL
LIN {X 0,Y 563.973,Z 843.44,A -85,B 0,C 180,E1 2714.296,E2 2714.296} C_VEL
LIN {X 0,Y 560.014,Z 843.44,A -85,B 0,C 180,E1 2716.041,E2 2716.041} C_VEL
LIN {X 0,Y 560.057,Z 843.44,A -85,B 0,C 180,E1 2720.503,E2 2720.503} C_VEL
LIN {X 0,Y 559.999,Z 843.44,A -85,B 0,C 180,E1 2725.539,E2 2725.539} C_VEL
LIN {X 0,Y 559.886,Z 843.44,A -85,B 0,C 180,E1 2730.802,E2 2730.802} C_VEL
LIN {X 0,Y 559.936,Z 843.44,A -85,B 0,C 180,E1 2736.361,E2 2736.361} C_VEL
LIN {X 0,Y 559.89,Z 843.44,A -85,B 0,C 180,E1 2742.359,E2 2742.359} C_VEL
LIN {X 0,Y 559.747,Z 843.44,A -85,B 0,C 180,E1 2747.626,E2 2747.626} C_VEL
LIN {X 0,Y 559.803,Z 843.595,A -85,B 0,C 180,E1 2752.977,E2 2752.977} C_VEL
LIN {X 0,Y 568.403,Z 861.65,A -85,B 0,C 180,E1 2753.905,E2 2753.905} C_VEL
LIN {X 0,Y 569.478,Z 866.57,A -85,B 0,C 180,E1 2754.059,E2 2754.059} C_VEL
LIN {X 0,Y 568.975,Z 914.121,A -85,B 0,C 180,E1 2754.964,E2 2754.964} C_VEL
LIN {X 0,Y 567.826,Z 954.929,A -85,B 0,C 180,E1 2756.347,E2 2756.347} C_VEL
LIN {X 0,Y 566.313,Z 997.076,A -85,B 0,C 180,E1 2758.501,E2 2758.501} C_VEL
LIN {X 0,Y 564.697,Z 1036.059,A -85,B 0,C 180,E1 2761.249,E2 2761.249} C_VEL
LIN {X 0,Y 563.3,Z 1070.247,A -85,B 0,C 180,E1 2764.407,E2 2764.407} C_VEL
LIN {X 0,Y 562.002,Z 1101.465,A -85,B 0,C 180,E1 2768.127,E2 2768.127} C_VEL
LIN {X 0,Y 561.246,Z 1126.535,A -85,B 0,C 180,E1 2771.989,E2 2771.989} C_VEL
LIN {X 0,Y 560.776,Z 1146.2,A -85,B 0,C 180,E1 2775.985,E2 2775.985} C_VEL
LIN {X 0,Y 560.422,Z 1161.399,A -85,B 0,C 180,E1 2780.315,E2 2780.315} C_VEL
LIN {X 0,Y 560.362,Z 1169.517,A -85,B 0,C 180,E1 2783.816,E2 2783.816} C_VEL
LIN {X 0,Y 560.394,Z 1173.637,A -85,B 0,C 180,E1 2786.913,E2 2786.913} C_VEL
LIN {X 0,Y 560.54,Z 1174.659,A -85,B 0,C 180,E1 2791.543,E2 2791.543} C_VEL
LIN {X 0,Y 560.362,Z 1169.517,A -85,B 0,C 180,E1 2796.184,E2 2796.184} C_VEL
LIN {X 0,Y 560.511,Z 1159.101,A -85,B 0,C 180,E1 2800.466,E2 2800.466} C_VEL
LIN {X 0,Y 560.736,Z 1144.015,A -85,B 0,C 180,E1 2804.515,E2 2804.515} C_VEL
LIN {X 0,Y 561.253,Z 1124.177,A -85,B 0,C 180,E1 2808.416,E2 2808.416} C_VEL
LIN {X 0,Y 562.111,Z 1098.032,A -85,B 0,C 180,E1 2812.331,E2 2812.331} C_VEL
LIN {X 0,Y 563.307,Z 1067.235,A -85,B 0,C 180,E1 2815.903,E2 2815.903} C_VEL
LIN {X 0,Y 564.828,Z 1032.917,A -85,B 0,C 180,E1 2818.999,E2 2818.999} C_VEL
LIN {X 0,Y 566.427,Z 995.585,A -85,B 0,C 180,E1 2821.583,E2 2821.583} C_VEL
LIN {X 0,Y 567.919,Z 954.06,A -85,B 0,C 180,E1 2823.684,E2 2823.684} C_VEL
LIN {X 0,Y 569.038,Z 909.669,A -85,B 0,C 180,E1 2825.156,E2 2825.156} C_VEL
LIN {X 0,Y 569.089,Z 862.717,A -85,B 0,C 180,E1 2826.028,E2 2826.028} C_VEL
LIN {X 0,Y 559.947,Z 845.04,A -85,B 0,C 180,E1 2826.989,E2 2826.989} C_VEL
LIN {X 0,Y 559.777,Z 843.44,A -85,B 0,C 180,E1 2827.077,E2 2827.077} C_VEL
LIN {X 0,Y 559.753,Z 843.44,A -85,B 0,C 180,E1 2833.293,E2 2833.293} C_VEL
LIN {X 0,Y 559.851,Z 843.44,A -85,B 0,C 180,E1 2839,E2 2839} C_VEL
LIN {X 0,Y 559.927,Z 843.44,A -85,B 0,C 180,E1 2843.95,E2 2843.95} C_VEL
LIN {X 0,Y 559.938,Z 843.44,A -85,B 0,C 180,E1 2849.586,E2 2849.586} C_VEL
LIN {X 0,Y 559.99,Z 843.44,A -85,B 0,C 180,E1 2854.46,E2 2854.46} C_VEL
LIN {X 0,Y 560.104,Z 843.44,A -85,B 0,C 180,E1 2860.555,E2 2860.555} C_VEL
LIN {X 0,Y 559.841,Z 843.44,A -85,B 0,C 180,E1 2865.961,E2 2865.961} C_VEL
LIN {X 0,Y 560.083,Z 843.44,A -85,B 0,C 180,E1 2870.697,E2 2870.697} C_VEL
LIN {X 0,Y 560.192,Z 843.44,A -85,B 0,C 180,E1 2875.365,E2 2875.365} C_VEL
LIN {X 0,Y 560.234,Z 843.44,A -85,B 0,C 180,E1 2880,E2 2880} C_VEL
LIN {X 0,Y 560.197,Z 843.44,A -85,B 0,C 180,E1 2884.67,E2 2884.67} C_VEL
LIN {X 0,Y 560.194,Z 843.44,A -85,B 0,C 180,E1 2889.301,E2 2889.301} C_VEL
LIN {X 0,Y 560.15,Z 843.44,A -85,B 0,C 180,E1 2894.111,E2 2894.111} C_VEL
LIN {X 0,Y 560.044,Z 843.44,A -85,B 0,C 180,E1 2899.428,E2 2899.428} C_VEL
LIN {X 0,Y 559.977,Z 843.44,A -85,B 0,C 180,E1 2903.841,E2 2903.841} C_VEL
LIN {X 0,Y 559.928,Z 843.44,A -85,B 0,C 180,E1 2909.018,E2 2909.018} C_VEL
LIN {X 0,Y 560.103,Z 843.44,A -85,B 0,C 180,E1 2914.454,E2 2914.454} C_VEL
LIN {X 0,Y 559.808,Z 843.44,A -85,B 0,C 180,E1 2920.309,E2 2920.309} C_VEL
LIN {X 0,Y 559.7,Z 843.44,A -85,B 0,C 180,E1 2925.493,E2 2925.493} C_VEL
LIN {X 0,Y 559.874,Z 843.44,A -85,B 0,C 180,E1 2931.407,E2 2931.407} C_VEL
LIN {X 0,Y 560.082,Z 843.44,A -85,B 0,C 180,E1 2933.402,E2 2933.402} C_VEL
LIN {X 0,Y 569.244,Z 863.187,A -85,B 0,C 180,E1 2934.437,E2 2934.437} C_VEL
LIN {X 0,Y 568.415,Z 905.703,A -85,B 0,C 180,E1 2935.575,E2 2935.575} C_VEL
LIN {X 0,Y 567.264,Z 943.802,A -85,B 0,C 180,E1 2937.184,E2 2937.184} C_VEL
LIN {X 0,Y 565.738,Z 981.959,A -85,B 0,C 180,E1 2939.417,E2 2939.417} C_VEL
LIN {X 0,Y 564.117,Z 1018.742,A -85,B 0,C 180,E1 2942.283,E2 2942.283} C_VEL
LIN {X 0,Y 562.741,Z 1051.474,A -85,B 0,C 180,E1 2945.589,E2 2945.589} C_VEL
LIN {X 0,Y 561.661,Z 1080.443,A -85,B 0,C 180,E1 2949.352,E2 2949.352} C_VEL
LIN {X 0,Y 560.913,Z 1104.344,A -85,B 0,C 180,E1 2953.391,E2 2953.391} C_VEL
LIN {X 0,Y 560.562,Z 1122.644,A -85,B 0,C 180,E1 2957.563,E2 2957.563} C_VEL
LIN {X 0,Y 560.375,Z 1134.585,A -85,B 0,C 180,E1 2961.483,E2 2961.483} C_VEL
LIN {X 0,Y 560.245,Z 1141.984,A -85,B 0,C 180,E1 2965.365,E2 2965.365} C_VEL
LIN {X 0,Y 560.285,Z 1144.677,A -85,B 0,C 180,E1 2968.457,E2 2968.457} C_VEL
LIN {X 0,Y 560.493,Z 1144.635,A -85,B 0,C 180,E1 2971.543,E2 2971.543} C_VEL
LIN {X 0,Y 560.434,Z 1141.311,A -85,B 0,C 180,E1 2974.989,E2 2974.989} C_VEL
LIN {X 0,Y 560.523,Z 1132.4,A -85,B 0,C 180,E1 2979.296,E2 2979.296} C_VEL
LIN {X 0,Y 560.689,Z 1117.677,A -85,B 0,C 180,E1 2983.621,E2 2983.621} C_VEL
LIN {X 0,Y 561.108,Z 1097.586,A -85,B 0,C 180,E1 2987.776,E2 2987.776} C_VEL
LIN {X 0,Y 561.979,Z 1072.614,A -85,B 0,C 180,E1 2991.667,E2 2991.667} C_VEL
LIN {X 0,Y 563.098,Z 1043.214,A -85,B 0,C 180,E1 2995.228,E2 2995.228} C_VEL
LIN {X 0,Y 564.577,Z 1009.412,A -85,B 0,C 180,E1 2998.423,E2 2998.423} C_VEL
LIN {X 0,Y 566.103,Z 973.276,A -85,B 0,C 180,E1 3001.059,E2 3001.059} C_VEL
LIN {X 0,Y 567.535,Z 935.824,A -85,B 0,C 180,E1 3003.114,E2 3003.114} C_VEL
LIN {X 0,Y 568.736,Z 895.664,A -85,B 0,C 180,E1 3004.666,E2 3004.666} C_VEL
LIN {X 0,Y 568.756,Z 862.374,A -85,B 0,C 180,E1 3005.523,E2 3005.523} C_VEL
LIN {X 0,Y 559.773,Z 843.44,A -85,B 0,C 180,E1 3006.572,E2 3006.572} C_VEL
LIN {X 0,Y 559.744,Z 843.44,A -85,B 0,C 180,E1 3012.374,E2 3012.374} C_VEL
LIN {X 0,Y 559.866,Z 843.44,A -85,B 0,C 180,E1 3017.639,E2 3017.639} C_VEL
LIN {X 0,Y 559.932,Z 843.44,A -85,B 0,C 180,E1 3023.949,E2 3023.949} C_VEL
LIN {X 0,Y 559.932,Z 843.44,A -85,B 0,C 180,E1 3029.587,E2 3029.587} C_VEL
LIN {X 0,Y 559.953,Z 843.44,A -85,B 0,C 180,E1 3034.459,E2 3034.459} C_VEL
LIN {X 0,Y 560.128,Z 843.44,A -85,B 0,C 180,E1 3040.547,E2 3040.547} C_VEL
LIN {X 0,Y 560.287,Z 843.44,A -85,B 0,C 180,E1 3045.973,E2 3045.973} C_VEL
LIN {X 0,Y 560.232,Z 843.44,A -85,B 0,C 180,E1 3052.26,E2 3052.26} C_VEL
LIN {X 0,Y 560.32,Z 843.44,A -85,B 0,C 180,E1 3056.913,E2 3056.913} C_VEL
LIN {X 0,Y 560.457,Z 843.44,A -85,B 0,C 180,E1 3061.543,E2 3061.543} C_VEL
LIN {X 0,Y 560.381,Z 843.44,A -85,B 0,C 180,E1 3066.183,E2 3066.183} C_VEL
LIN {X 0,Y 560.022,Z 843.44,A -85,B 0,C 180,E1 3072.565,E2 3072.565} C_VEL
LIN {X 0,Y 560.014,Z 843.44,A -85,B 0,C 180,E1 3076.041,E2 3076.041} C_VEL
LIN {X 0,Y 556.036,Z 843.44,A -85,B 0,C 180,E1 3077.785,E2 3077.785} C_VEL
LIN {X 0,Y 552.064,Z 843.44,A -85,B 0,C 180,E1 3079.554,E2 3079.554} C_VEL
LIN {X 0,Y 552.104,Z 843.44,A -85,B 0,C 180,E1 3085.584,E2 3085.584} C_VEL
LIN {X 0,Y 551.896,Z 843.44,A -85,B 0,C 180,E1 3091.298,E2 3091.298} C_VEL
LIN {X 0,Y 551.961,Z 843.44,A -85,B 0,C 180,E1 3097.549,E2 3097.549} C_VEL
LIN {X 0,Y 551.965,Z 843.44,A -85,B 0,C 180,E1 3103.114,E2 3103.114} C_VEL
LIN {X 0,Y 551.862,Z 843.44,A -85,B 0,C 180,E1 3108.985,E2 3108.985} C_VEL
LIN {X 0,Y 551.892,Z 844.114,A -85,B 0,C 180,E1 3112.364,E2 3112.364} C_VEL
LIN {X 0,Y 563.077,Z 866.83,A -85,B 0,C 180,E1 3113.59,E2 3113.59} C_VEL
LIN {X 0,Y 562.51,Z 914.22,A -85,B 0,C 180,E1 3114.504,E2 3114.504} C_VEL
LIN {X 0,Y 561.121,Z 955.717,A -85,B 0,C 180,E1 3115.927,E2 3115.927} C_VEL
LIN {X 0,Y 559.381,Z 997.074,A -85,B 0,C 180,E1 3118.065,E2 3118.065} C_VEL
LIN {X 0,Y 557.525,Z 1036.057,A -85,B 0,C 180,E1 3120.844,E2 3120.844} C_VEL
LIN {X 0,Y 555.863,Z 1071.03,A -85,B 0,C 180,E1 3124.128,E2 3124.128} C_VEL
LIN {X 0,Y 554.354,Z 1101.863,A -85,B 0,C 180,E1 3127.866,E2 3127.866} C_VEL
LIN {X 0,Y 553.454,Z 1127.632,A -85,B 0,C 180,E1 3131.932,E2 3131.932} C_VEL
LIN {X 0,Y 552.864,Z 1147.853,A -85,B 0,C 180,E1 3136.183,E2 3136.183} C_VEL
LIN {X 0,Y 552.596,Z 1160.807,A -85,B 0,C 180,E1 3139.972,E2 3139.972} C_VEL
LIN {X 0,Y 552.47,Z 1169.517,A -85,B 0,C 180,E1 3143.728,E2 3143.728} C_VEL
LIN {X 0,Y 552.512,Z 1173.637,A -85,B 0,C 180,E1 3146.869,E2 3146.869} C_VEL
LIN {X 0,Y 552.636,Z 1174.659,A -85,B 0,C 180,E1 3151.565,E2 3151.565} C_VEL
LIN {X 0,Y 552.471,Z 1169.517,A -85,B 0,C 180,E1 3156.273,E2 3156.273} C_VEL
LIN {X 0,Y 552.686,Z 1159.097,A -85,B 0,C 180,E1 3160.617,E2 3160.617} C_VEL
LIN {X 0,Y 552.999,Z 1142.707,A -85,B 0,C 180,E1 3165.025,E2 3165.025} C_VEL
LIN {X 0,Y 553.632,Z 1121.76,A -85,B 0,C 180,E1 3169.092,E2 3169.092} C_VEL
LIN {X 0,Y 554.59,Z 1096.799,A -85,B 0,C 180,E1 3172.814,E2 3172.814} C_VEL
LIN {X 0,Y 555.983,Z 1065.886,A -85,B 0,C 180,E1 3176.41,E2 3176.41} C_VEL
LIN {X 0,Y 557.738,Z 1031.611,A -85,B 0,C 180,E1 3179.509,E2 3179.509} C_VEL
LIN {X 0,Y 559.585,Z 993.954,A -85,B 0,C 180,E1 3182.114,E2 3182.114} C_VEL
LIN {X 0,Y 561.261,Z 953.94,A -85,B 0,C 180,E1 3184.143,E2 3184.143} C_VEL
LIN {X 0,Y 562.548,Z 909.375,A -85,B 0,C 180,E1 3185.63,E2 3185.63} C_VEL
LIN {X 0,Y 562.571,Z 865.537,A -85,B 0,C 180,E1 3186.468,E2 3186.468} C_VEL
LIN {X 0,Y 551.866,Z 843.44,A -85,B 0,C 180,E1 3187.727,E2 3187.727} C_VEL
LIN {X 0,Y 551.844,Z 843.44,A -85,B 0,C 180,E1 3193.128,E2 3193.128} C_VEL
LIN {X 0,Y 551.966,Z 843.44,A -85,B 0,C 180,E1 3198.996,E2 3198.996} C_VEL
LIN {X 0,Y 551.914,Z 843.44,A -85,B 0,C 180,E1 3205.11,E2 3205.11} C_VEL
LIN {X 0,Y 551.951,Z 843.44,A -85,B 0,C 180,E1 3211.03,E2 3211.03} C_VEL
LIN {X 0,Y 552.007,Z 843.44,A -85,B 0,C 180,E1 3215.793,E2 3215.793} C_VEL
LIN {X 0,Y 552.222,Z 843.44,A -85,B 0,C 180,E1 3220.858,E2 3220.858} C_VEL
LIN {X 0,Y 551.94,Z 843.44,A -85,B 0,C 180,E1 3225.756,E2 3225.756} C_VEL
LIN {X 0,Y 552.171,Z 843.44,A -85,B 0,C 180,E1 3230.563,E2 3230.563} C_VEL
LIN {X 0,Y 552.326,Z 843.44,A -85,B 0,C 180,E1 3235.299,E2 3235.299} C_VEL
LIN {X 0,Y 552.337,Z 843.44,A -85,B 0,C 180,E1 3240,E2 3240} C_VEL
LIN {X 0,Y 552.319,Z 843.44,A -85,B 0,C 180,E1 3244.701,E2 3244.701} C_VEL
LIN {X 0,Y 552.168,Z 843.44,A -85,B 0,C 180,E1 3250.313,E2 3250.313} C_VEL
LIN {X 0,Y 552.09,Z 843.44,A -85,B 0,C 180,E1 3255.862,E2 3255.862} C_VEL
LIN {X 0,Y 552.07,Z 843.44,A -85,B 0,C 180,E1 3261.666,E2 3261.666} C_VEL
LIN {X 0,Y 551.968,Z 843.44,A -85,B 0,C 180,E1 3267.693,E2 3267.693} C_VEL
LIN {X 0,Y 552.16,Z 843.44,A -85,B 0,C 180,E1 3273.131,E2 3273.131} C_VEL
LIN {X 0,Y 551.955,Z 843.44,A -85,B 0,C 180,E1 3278.96,E2 3278.96} C_VEL
LIN {X 0,Y 551.796,Z 843.44,A -85,B 0,C 180,E1 3284.681,E2 3284.681} C_VEL
LIN {X 0,Y 551.911,Z 843.44,A -85,B 0,C 180,E1 3289.954,E2 3289.954} C_VEL
LIN {X 0,Y 552.138,Z 843.44,A -85,B 0,C 180,E1 3292.789,E2 3292.789} C_VEL
LIN {X 0,Y 562.808,Z 866.254,A -85,B 0,C 180,E1 3294.027,E2 3294.027} C_VEL
LIN {X 0,Y 561.79,Z 909.455,A -85,B 0,C 180,E1 3295.247,E2 3295.247} C_VEL
LIN {X 0,Y 560.268,Z 949.451,A -85,B 0,C 180,E1 3297.029,E2 3297.029} C_VEL
LIN {X 0,Y 558.578,Z 985.537,A -85,B 0,C 180,E1 3299.246,E2 3299.246} C_VEL
LIN {X 0,Y 556.736,Z 1021.451,A -85,B 0,C 180,E1 3302.143,E2 3302.143} C_VEL
LIN {X 0,Y 555.107,Z 1054.018,A -85,B 0,C 180,E1 3305.542,E2 3305.542} C_VEL
LIN {X 0,Y 553.937,Z 1081.777,A -85,B 0,C 180,E1 3309.259,E2 3309.259} C_VEL
LIN {X 0,Y 553.144,Z 1103.902,A -85,B 0,C 180,E1 3313.059,E2 3313.059} C_VEL
LIN {X 0,Y 552.748,Z 1121.111,A -85,B 0,C 180,E1 3316.984,E2 3316.984} C_VEL
LIN {X 0,Y 552.49,Z 1132.652,A -85,B 0,C 180,E1 3320.568,E2 3320.568} C_VEL
LIN {X 0,Y 552.386,Z 1140.799,A -85,B 0,C 180,E1 3324.513,E2 3324.513} C_VEL
LIN {X 0,Y 552.394,Z 1144.677,A -85,B 0,C 180,E1 3328.434,E2 3328.434} C_VEL
LIN {X 0,Y 552.587,Z 1144.635,A -85,B 0,C 180,E1 3331.565,E2 3331.565} C_VEL
LIN {X 0,Y 552.491,Z 1140.662,A -85,B 0,C 180,E1 3335.485,E2 3335.485} C_VEL
LIN {X 0,Y 552.62,Z 1132.402,A -85,B 0,C 180,E1 3339.43,E2 3339.43} C_VEL
LIN {X 0,Y 552.845,Z 1117.681,A -85,B 0,C 180,E1 3343.818,E2 3343.818} C_VEL
LIN {X 0,Y 553.361,Z 1097.392,A -85,B 0,C 180,E1 3348.071,E2 3348.071} C_VEL
LIN {X 0,Y 554.338,Z 1071.602,A -85,B 0,C 180,E1 3352.127,E2 3352.127} C_VEL
LIN {X 0,Y 555.838,Z 1040.631,A -85,B 0,C 180,E1 3355.874,E2 3355.874} C_VEL
LIN {X 0,Y 557.609,Z 1005.542,A -85,B 0,C 180,E1 3359.151,E2 3359.151} C_VEL
LIN {X 0,Y 559.448,Z 967.899,A -85,B 0,C 180,E1 3361.831,E2 3361.831} C_VEL
LIN {X 0,Y 561.115,Z 929.414,A -85,B 0,C 180,E1 3363.851,E2 3363.851} C_VEL
LIN {X 0,Y 562.41,Z 891.315,A -85,B 0,C 180,E1 3365.246,E2 3365.246} C_VEL
LIN {X 0,Y 562.524,Z 865.779,A -85,B 0,C 180,E1 3365.915,E2 3365.915} C_VEL
LIN {X 0,Y 551.837,Z 843.44,A -85,B 0,C 180,E1 3367.229,E2 3367.229} C_VEL
LIN {X 0,Y 551.835,Z 843.44,A -85,B 0,C 180,E1 3373.128,E2 3373.128} C_VEL
LIN {X 0,Y 551.954,Z 843.44,A -85,B 0,C 180,E1 3378.996,E2 3378.996} C_VEL
LIN {X 0,Y 551.897,Z 843.44,A -85,B 0,C 180,E1 3385.111,E2 3385.111} C_VEL
LIN {X 0,Y 551.949,Z 843.44,A -85,B 0,C 180,E1 3391.03,E2 3391.03} C_VEL
LIN {X 0,Y 551.994,Z 843.44,A -85,B 0,C 180,E1 3395.792,E2 3395.792} C_VEL
LIN {X 0,Y 552.244,Z 843.44,A -85,B 0,C 180,E1 3400.859,E2 3400.859} C_VEL
LIN {X 0,Y 552.373,Z 843.44,A -85,B 0,C 180,E1 3405.768,E2 3405.768} C_VEL
LIN {X 0,Y 552.318,Z 843.44,A -85,B 0,C 180,E1 3412.149,E2 3412.149} C_VEL
LIN {X 0,Y 552.42,Z 843.44,A -85,B 0,C 180,E1 3416.868,E2 3416.868} C_VEL
LIN {X 0,Y 552.549,Z 843.44,A -85,B 0,C 180,E1 3421.565,E2 3421.565} C_VEL
LIN {X 0,Y 552.45,Z 843.44,A -85,B 0,C 180,E1 3426.273,E2 3426.273} C_VEL
LIN {X 0,Y 552.123,Z 843.44,A -85,B 0,C 180,E1 3432.629,E2 3432.629} C_VEL
LIN {X 0,Y 552.106,Z 843.44,A -85,B 0,C 180,E1 3437.496,E2 3437.496} C_VEL
LIN {X 0,Y 552.064,Z 843.44,A -85,B 0,C 180,E1 3439.554,E2 3439.554} C_VEL
LIN {X 0,Y 548.055,Z 843.44,A -85,B 0,C 180,E1 3441.324,E2 3441.324} C_VEL
LIN {X 0,Y 544.06,Z 843.44,A -85,B 0,C 180,E1 3443.12,E2 3443.12} C_VEL
LIN {X 0,Y 544.039,Z 843.44,A -85,B 0,C 180,E1 3448.133,E2 3448.133} C_VEL
LIN {X 0,Y 543.92,Z 843.44,A -85,B 0,C 180,E1 3453.7,E2 3453.7} C_VEL
LIN {X 0,Y 544.021,Z 843.44,A -85,B 0,C 180,E1 3459.639,E2 3459.639} C_VEL
LIN {X 0,Y 544.01,Z 843.44,A -85,B 0,C 180,E1 3463.903,E2 3463.903} C_VEL
LIN {X 0,Y 543.907,Z 843.44,A -85,B 0,C 180,E1 3470.349,E2 3470.349} C_VEL
LIN {X 0,Y 543.966,Z 843.44,A -85,B 0,C 180,E1 3471.697,E2 3471.697} C_VEL
LIN {X 0,Y 548.517,Z 853.575,A -85,B 0,C 180,E1 3472.245,E2 3472.245} C_VEL
LIN {X 0,Y 556.694,Z 869.66,A -85,B 0,C 180,E1 3473.148,E2 3473.148} C_VEL
LIN {X 0,Y 556.019,Z 914.972,A -85,B 0,C 180,E1 3474.048,E2 3474.048} C_VEL
LIN {X 0,Y 554.444,Z 956.62,A -85,B 0,C 180,E1 3475.503,E2 3475.503} C_VEL
LIN {X 0,Y 552.424,Z 998.375,A -85,B 0,C 180,E1 3477.703,E2 3477.703} C_VEL
LIN {X 0,Y 550.377,Z 1036.054,A -85,B 0,C 180,E1 3480.428,E2 3480.428} C_VEL
LIN {X 0,Y 548.455,Z 1071.029,A -85,B 0,C 180,E1 3483.752,E2 3483.752} C_VEL
LIN {X 0,Y 546.793,Z 1101.864,A -85,B 0,C 180,E1 3487.543,E2 3487.543} C_VEL
LIN {X 0,Y 545.723,Z 1127.634,A -85,B 0,C 180,E1 3491.667,E2 3491.667} C_VEL
LIN {X 0,Y 545.027,Z 1148.106,A -85,B 0,C 180,E1 3496.047,E2 3496.047} C_VEL
LIN {X 0,Y 544.621,Z 1162.53,A -85,B 0,C 180,E1 3500.431,E2 3500.431} C_VEL
LIN {X 0,Y 544.514,Z 1170.731,A -85,B 0,C 180,E1 3504.434,E2 3504.434} C_VEL
LIN {X 0,Y 544.479,Z 1174.659,A -85,B 0,C 180,E1 3508.412,E2 3508.412} C_VEL
LIN {X 0,Y 544.732,Z 1174.659,A -85,B 0,C 180,E1 3511.588,E2 3511.588} C_VEL
LIN {X 0,Y 544.608,Z 1169.517,A -85,B 0,C 180,E1 3516.364,E2 3516.364} C_VEL
LIN {X 0,Y 544.784,Z 1159.657,A -85,B 0,C 180,E1 3520.577,E2 3520.577} C_VEL
LIN {X 0,Y 545.115,Z 1144.459,A -85,B 0,C 180,E1 3524.837,E2 3524.837} C_VEL
LIN {X 0,Y 545.793,Z 1124.173,A -85,B 0,C 180,E1 3528.958,E2 3528.958} C_VEL
LIN {X 0,Y 546.952,Z 1098.392,A -85,B 0,C 180,E1 3532.936,E2 3532.936} C_VEL
LIN {X 0,Y 548.541,Z 1067.589,A -85,B 0,C 180,E1 3536.617,E2 3536.617} C_VEL
LIN {X 0,Y 550.567,Z 1032.656,A -85,B 0,C 180,E1 3539.847,E2 3539.847} C_VEL
LIN {X 0,Y 552.694,Z 994.954,A -85,B 0,C 180,E1 3542.502,E2 3542.502} C_VEL
LIN {X 0,Y 554.622,Z 954.055,A -85,B 0,C 180,E1 3544.605,E2 3544.605} C_VEL
LIN {X 0,Y 556.099,Z 911.052,A -85,B 0,C 180,E1 3546.065,E2 3546.065} C_VEL
LIN {X 0,Y 556.117,Z 868.099,A -85,B 0,C 180,E1 3546.921,E2 3546.921} C_VEL
LIN {X 0,Y 544.055,Z 844.766,A -85,B 0,C 180,E1 3548.265,E2 3548.265} C_VEL
LIN {X 0,Y 543.928,Z 843.44,A -85,B 0,C 180,E1 3548.351,E2 3548.351} C_VEL
LIN {X 0,Y 543.935,Z 843.44,A -85,B 0,C 180,E1 3553.913,E2 3553.913} C_VEL
LIN {X 0,Y 544.033,Z 843.44,A -85,B 0,C 180,E1 3558.497,E2 3558.497} C_VEL
LIN {X 0,Y 543.962,Z 843.44,A -85,B 0,C 180,E1 3564.37,E2 3564.37} C_VEL
LIN {X 0,Y 543.991,Z 843.44,A -85,B 0,C 180,E1 3570.047,E2 3570.047} C_VEL
LIN {X 0,Y 544.106,Z 843.44,A -85,B 0,C 180,E1 3575.418,E2 3575.418} C_VEL
LIN {X 0,Y 544.282,Z 843.44,A -85,B 0,C 180,E1 3580.568,E2 3580.568} C_VEL
LIN {X 0,Y 544.01,Z 843.44,A -85,B 0,C 180,E1 3586.134,E2 3586.134} C_VEL
LIN {X 0,Y 544.289,Z 843.44,A -85,B 0,C 180,E1 3590.425,E2 3590.425} C_VEL
LIN {X 0,Y 544.439,Z 843.44,A -85,B 0,C 180,E1 3595.23,E2 3595.23} C_VEL
LIN {X 0,Y 544.436,Z 843.44,A -85,B 0,C 180,E1 3600,E2 3600} C_VEL
LIN {X 0,Y 544.425,Z 843.44,A -85,B 0,C 180,E1 3604.769,E2 3604.769} C_VEL
LIN {X 0,Y 544.36,Z 843.44,A -85,B 0,C 180,E1 3609.574,E2 3609.574} C_VEL
LIN {X 0,Y 544.312,Z 843.44,A -85,B 0,C 180,E1 3614.448,E2 3614.448} C_VEL
LIN {X 0,Y 544.22,Z 843.44,A -85,B 0,C 180,E1 3619.48,E2 3619.48} C_VEL
LIN {X 0,Y 544.082,Z 843.44,A -85,B 0,C 180,E1 3624.583,E2 3624.583} C_VEL
LIN {X 0,Y 544.06,Z 843.44,A -85,B 0,C 180,E1 3630.703,E2 3630.703} C_VEL
LIN {X 0,Y 544.151,Z 843.44,A -85,B 0,C 180,E1 3635.615,E2 3635.615} C_VEL
LIN {X 0,Y 543.963,Z 843.44,A -85,B 0,C 180,E1 3641.74,E2 3641.74} C_VEL
LIN {X 0,Y 544.007,Z 843.44,A -85,B 0,C 180,E1 3648.497,E2 3648.497} C_VEL
LIN {X 0,Y 544.157,Z 843.44,A -85,B 0,C 180,E1 3652.157,E2 3652.157} C_VEL
LIN {X 0,Y 548.874,Z 853.73,A -85,B 0,C 180,E1 3652.724,E2 3652.724} C_VEL
LIN {X 0,Y 556.35,Z 869.096,A -85,B 0,C 180,E1 3653.613,E2 3653.613} C_VEL
LIN {X 0,Y 555.14,Z 911.535,A -85,B 0,C 180,E1 3654.853,E2 3654.853} C_VEL
LIN {X 0,Y 553.388,Z 952.216,A -85,B 0,C 180,E1 3656.72,E2 3656.72} C_VEL
LIN {X 0,Y 551.315,Z 990.644,A -85,B 0,C 180,E1 3659.181,E2 3659.181} C_VEL
LIN {X 0,Y 549.195,Z 1027.196,A -85,B 0,C 180,E1 3662.288,E2 3662.288} C_VEL
LIN {X 0,Y 547.326,Z 1060.709,A -85,B 0,C 180,E1 3666.004,E2 3666.004} C_VEL
LIN {X 0,Y 545.996,Z 1088.337,A -85,B 0,C 180,E1 3669.992,E2 3669.992} C_VEL
LIN {X 0,Y 545.182,Z 1111.149,A -85,B 0,C 180,E1 3674.343,E2 3674.343} C_VEL
LIN {X 0,Y 544.843,Z 1128.047,A -85,B 0,C 180,E1 3678.821,E2 3678.821} C_VEL
LIN {X 0,Y 544.682,Z 1138.051,A -85,B 0,C 180,E1 3682.838,E2 3682.838} C_VEL
LIN {X 0,Y 544.608,Z 1143.674,A -85,B 0,C 180,E1 3686.823,E2 3686.823} C_VEL
LIN {X 0,Y 544.682,Z 1144.636,A -85,B 0,C 180,E1 3691.587,E2 3691.587} C_VEL
LIN {X 0,Y 544.607,Z 1140.663,A -85,B 0,C 180,E1 3695.565,E2 3695.565} C_VEL
LIN {X 0,Y 544.715,Z 1132.403,A -85,B 0,C 180,E1 3699.568,E2 3699.568} C_VEL
LIN {X 0,Y 544.978,Z 1118.074,A -85,B 0,C 180,E1 3703.918,E2 3703.918} C_VEL
LIN {X 0,Y 545.572,Z 1098.492,A -85,B 0,C 180,E1 3708.129,E2 3708.129} C_VEL
LIN {X 0,Y 546.633,Z 1074.065,A -85,B 0,C 180,E1 3712.098,E2 3712.098} C_VEL
LIN {X 0,Y 548.145,Z 1045.537,A -85,B 0,C 180,E1 3715.702,E2 3715.702} C_VEL
LIN {X 0,Y 550.037,Z 1012.563,A -85,B 0,C 180,E1 3718.964,E2 3718.964} C_VEL
LIN {X 0,Y 552.097,Z 975.936,A -85,B 0,C 180,E1 3721.757,E2 3721.757} C_VEL
LIN {X 0,Y 554.07,Z 938.027,A -85,B 0,C 180,E1 3723.92,E2 3723.92} C_VEL
LIN {X 0,Y 555.721,Z 896.202,A -85,B 0,C 180,E1 3725.582,E2 3725.582} C_VEL
LIN {X 0,Y 555.815,Z 868.094,A -85,B 0,C 180,E1 3726.362,E2 3726.362} C_VEL
LIN {X 0,Y 543.936,Z 844.243,A -85,B 0,C 180,E1 3727.746,E2 3727.746} C_VEL
LIN {X 0,Y 543.913,Z 843.44,A -85,B 0,C 180,E1 3731.747,E2 3731.747} C_VEL
LIN {X 0,Y 544.024,Z 843.44,A -85,B 0,C 180,E1 3738.265,E2 3738.265} C_VEL
LIN {X 0,Y 543.954,Z 843.44,A -85,B 0,C 180,E1 3744.37,E2 3744.37} C_VEL
LIN {X 0,Y 543.984,Z 843.44,A -85,B 0,C 180,E1 3750.046,E2 3750.046} C_VEL
LIN {X 0,Y 544.074,Z 843.44,A -85,B 0,C 180,E1 3756.244,E2 3756.244} C_VEL
LIN {X 0,Y 544.307,Z 843.44,A -85,B 0,C 180,E1 3760.569,E2 3760.569} C_VEL
LIN {X 0,Y 544.457,Z 843.44,A -85,B 0,C 180,E1 3765.943,E2 3765.943} C_VEL
LIN {X 0,Y 544.402,Z 843.44,A -85,B 0,C 180,E1 3772.034,E2 3772.034} C_VEL
LIN {X 0,Y 544.512,Z 843.44,A -85,B 0,C 180,E1 3776.823,E2 3776.823} C_VEL
LIN {X 0,Y 544.638,Z 843.44,A -85,B 0,C 180,E1 3781.588,E2 3781.588} C_VEL
LIN {X 0,Y 544.521,Z 843.44,A -85,B 0,C 180,E1 3786.364,E2 3786.364} C_VEL
LIN {X 0,Y 544.336,Z 843.44,A -85,B 0,C 180,E1 3791.189,E2 3791.189} C_VEL
LIN {X 0,Y 544.23,Z 843.44,A -85,B 0,C 180,E1 3796.097,E2 3796.097} C_VEL
LIN {X 0,Y 544.179,Z 843.44,A -85,B 0,C 180,E1 3801.13,E2 3801.13} C_VEL
LIN {X 0,Y 544.06,Z 843.44,A -85,B 0,C 180,E1 3803.12,E2 3803.12} C_VEL
LIN {X 0,Y 542.772,Z 843.44,A -85,B 0,C 180,E1 3804.033,E2 3804.033} C_VEL
LIN {X 0,Y 536.232,Z 843.44,A -85,B 0,C 180,E1 3806.518,E2 3806.518} C_VEL
LIN {X 0,Y 536.162,Z 843.44,A -85,B 0,C 180,E1 3806.753,E2 3806.753} C_VEL
LIN {X 0,Y 536.025,Z 843.44,A -85,B 0,C 180,E1 3812.376,E2 3812.376} C_VEL
LIN {X 0,Y 536.133,Z 843.44,A -85,B 0,C 180,E1 3818.257,E2 3818.257} C_VEL
LIN {X 0,Y 535.987,Z 843.44,A -85,B 0,C 180,E1 3824.735,E2 3824.735} C_VEL
LIN {X 0,Y 536.025,Z 843.496,A -85,B 0,C 180,E1 3831.034,E2 3831.034} C_VEL
LIN {X 0,Y 540.536,Z 853.421,A -85,B 0,C 180,E1 3831.584,E2 3831.584} C_VEL
LIN {X 0,Y 550.251,Z 871.942,A -85,B 0,C 180,E1 3832.681,E2 3832.681} C_VEL
LIN {X 0,Y 549.51,Z 916.877,A -85,B 0,C 180,E1 3833.614,E2 3833.614} C_VEL
LIN {X 0,Y 547.823,Z 956.839,A -85,B 0,C 180,E1 3835.037,E2 3835.037} C_VEL
LIN {X 0,Y 545.648,Z 997.45,A -85,B 0,C 180,E1 3837.188,E2 3837.188} C_VEL
LIN {X 0,Y 543.283,Z 1036.051,A -85,B 0,C 180,E1 3840.002,E2 3840.002} C_VEL
LIN {X 0,Y 541.081,Z 1070.733,A -85,B 0,C 180,E1 3843.332,E2 3843.332} C_VEL
LIN {X 0,Y 539.221,Z 1101.171,A -85,B 0,C 180,E1 3847.108,E2 3847.108} C_VEL
LIN {X 0,Y 538.02,Z 1126.54,A -85,B 0,C 180,E1 3851.183,E2 3851.183} C_VEL
LIN {X 0,Y 537.312,Z 1146.196,A -85,B 0,C 180,E1 3855.359,E2 3855.359} C_VEL
LIN {X 0,Y 536.909,Z 1160.672,A -85,B 0,C 180,E1 3859.628,E2 3859.628} C_VEL
LIN {X 0,Y 536.713,Z 1169.517,A -85,B 0,C 180,E1 3863.543,E2 3863.543} C_VEL
LIN {X 0,Y 536.703,Z 1173.637,A -85,B 0,C 180,E1 3866.777,E2 3866.777} C_VEL
LIN {X 0,Y 536.856,Z 1174.659,A -85,B 0,C 180,E1 3871.611,E2 3871.611} C_VEL
LIN {X 0,Y 536.715,Z 1169.517,A -85,B 0,C 180,E1 3876.457,E2 3876.457} C_VEL
LIN {X 0,Y 536.935,Z 1159.592,A -85,B 0,C 180,E1 3880.756,E2 3880.756} C_VEL
LIN {X 0,Y 537.29,Z 1144.46,A -85,B 0,C 180,E1 3885.058,E2 3885.058} C_VEL
LIN {X 0,Y 538.076,Z 1124.171,A -85,B 0,C 180,E1 3889.24,E2 3889.24} C_VEL
LIN {X 0,Y 539.421,Z 1098.391,A -85,B 0,C 180,E1 3893.275,E2 3893.275} C_VEL
LIN {X 0,Y 541.255,Z 1067.181,A -85,B 0,C 180,E1 3897.048,E2 3897.048} C_VEL
LIN {X 0,Y 543.466,Z 1033.359,A -85,B 0,C 180,E1 3900.218,E2 3900.218} C_VEL
LIN {X 0,Y 545.817,Z 995.3,A -85,B 0,C 180,E1 3902.941,E2 3902.941} C_VEL
LIN {X 0,Y 548.03,Z 953.197,A -85,B 0,C 180,E1 3905.119,E2 3905.119} C_VEL
LIN {X 0,Y 549.737,Z 909.275,A -85,B 0,C 180,E1 3906.596,E2 3906.596} C_VEL
LIN {X 0,Y 549.945,Z 871.397,A -85,B 0,C 180,E1 3907.352,E2 3907.352} C_VEL
LIN {X 0,Y 536.154,Z 844.97,A -85,B 0,C 180,E1 3908.93,E2 3908.93} C_VEL
LIN {X 0,Y 536.003,Z 843.44,A -85,B 0,C 180,E1 3909.081,E2 3909.081} C_VEL
LIN {X 0,Y 535.988,Z 843.44,A -85,B 0,C 180,E1 3915.266,E2 3915.266} C_VEL
LIN {X 0,Y 536.127,Z 843.44,A -85,B 0,C 180,E1 3921.742,E2 3921.742} C_VEL
LIN {X 0,Y 536.055,Z 843.44,A -85,B 0,C 180,E1 3927.667,E2 3927.667} C_VEL
LIN {X 0,Y 536.141,Z 843.44,A -85,B 0,C 180,E1 3933.236,E2 3933.236} C_VEL
LIN {X 0,Y 536.24,Z 843.44,A -85,B 0,C 180,E1 3938.542,E2 3938.542} C_VEL
LIN {X 0,Y 536.323,Z 843.44,A -85,B 0,C 180,E1 3943.659,E2 3943.659} C_VEL
LIN {X 0,Y 536.369,Z 843.44,A -85,B 0,C 180,E1 3950.282,E2 3950.282} C_VEL
LIN {X 0,Y 536.535,Z 843.44,A -85,B 0,C 180,E1 3955.16,E2 3955.16} C_VEL
LIN {X 0,Y 536.543,Z 843.44,A -85,B 0,C 180,E1 3960,E2 3960} C_VEL
LIN {X 0,Y 536.512,Z 843.44,A -85,B 0,C 180,E1 3964.84,E2 3964.84} C_VEL
LIN {X 0,Y 536.386,Z 843.44,A -85,B 0,C 180,E1 3970.05,E2 3970.05} C_VEL
LIN {X 0,Y 536.372,Z 843.44,A -85,B 0,C 180,E1 3974.666,E2 3974.666} C_VEL
LIN {X 0,Y 536.31,Z 843.44,A -85,B 0,C 180,E1 3979.732,E2 3979.732} C_VEL
LIN {X 0,Y 536.077,Z 843.44,A -85,B 0,C 180,E1 3985.74,E2 3985.74} C_VEL
LIN {X 0,Y 536.145,Z 843.44,A -85,B 0,C 180,E1 3990.438,E2 3990.438} C_VEL
LIN {X 0,Y 536.222,Z 843.44,A -85,B 0,C 180,E1 3996.224,E2 3996.224} C_VEL
LIN {X 0,Y 535.945,Z 843.44,A -85,B 0,C 180,E1 4002.51,E2 4002.51} C_VEL
LIN {X 0,Y 535.988,Z 843.44,A -85,B 0,C 180,E1 4007.492,E2 4007.492} C_VEL
LIN {X 0,Y 536.185,Z 843.44,A -85,B 0,C 180,E1 4011.472,E2 4011.472} C_VEL
LIN {X 0,Y 542.965,Z 857.748,A -85,B 0,C 180,E1 4012.327,E2 4012.327} C_VEL
LIN {X 0,Y 549.897,Z 871.714,A -85,B 0,C 180,E1 4013.182,E2 4013.182} C_VEL
LIN {X 0,Y 548.576,Z 912.539,A -85,B 0,C 180,E1 4014.414,E2 4014.414} C_VEL
LIN {X 0,Y 546.617,Z 952.883,A -85,B 0,C 180,E1 4016.291,E2 4016.291} C_VEL
LIN {X 0,Y 544.251,Z 991.676,A -85,B 0,C 180,E1 4018.816,E2 4018.816} C_VEL
LIN {X 0,Y 541.915,Z 1027.889,A -85,B 0,C 180,E1 4021.952,E2 4021.952} C_VEL
LIN {X 0,Y 539.808,Z 1060.768,A -85,B 0,C 180,E1 4025.657,E2 4025.657} C_VEL
LIN {X 0,Y 538.321,Z 1088.335,A -85,B 0,C 180,E1 4029.694,E2 4029.694} C_VEL
LIN {X 0,Y 537.367,Z 1111.148,A -85,B 0,C 180,E1 4034.11,E2 4034.11} C_VEL
LIN {X 0,Y 536.97,Z 1128.044,A -85,B 0,C 180,E1 4038.655,E2 4038.655} C_VEL
LIN {X 0,Y 536.785,Z 1138.05,A -85,B 0,C 180,E1 4042.732,E2 4042.732} C_VEL
LIN {X 0,Y 536.709,Z 1143.673,A -85,B 0,C 180,E1 4046.776,E2 4046.776} C_VEL
LIN {X 0,Y 536.806,Z 1144.636,A -85,B 0,C 180,E1 4051.611,E2 4051.611} C_VEL
LIN {X 0,Y 536.713,Z 1140.664,A -85,B 0,C 180,E1 4055.647,E2 4055.647} C_VEL
LIN {X 0,Y 536.819,Z 1132.405,A -85,B 0,C 180,E1 4059.71,E2 4059.71} C_VEL
LIN {X 0,Y 537.119,Z 1118.467,A -85,B 0,C 180,E1 4064.021,E2 4064.021} C_VEL
LIN {X 0,Y 537.789,Z 1099.593,A -85,B 0,C 180,E1 4068.189,E2 4068.189} C_VEL
LIN {X 0,Y 538.939,Z 1075.883,A -85,B 0,C 180,E1 4072.162,E2 4072.162} C_VEL
LIN {X 0,Y 540.648,Z 1047.513,A -85,B 0,C 180,E1 4075.856,E2 4075.856} C_VEL
LIN {X 0,Y 542.78,Z 1014.317,A -85,B 0,C 180,E1 4079.229,E2 4079.229} C_VEL
LIN {X 0,Y 545.137,Z 977.099,A -85,B 0,C 180,E1 4082.131,E2 4082.131} C_VEL
LIN {X 0,Y 547.379,Z 939.038,A -85,B 0,C 180,E1 4084.342,E2 4084.342} C_VEL
LIN {X 0,Y 549.192,Z 897.768,A -85,B 0,C 180,E1 4086.014,E2 4086.014} C_VEL
LIN {X 0,Y 549.649,Z 871.701,A -85,B 0,C 180,E1 4086.747,E2 4086.747} C_VEL
LIN {X 0,Y 536.066,Z 844.733,A -85,B 0,C 180,E1 4088.392,E2 4088.392} C_VEL
LIN {X 0,Y 535.938,Z 843.44,A -85,B 0,C 180,E1 4088.453,E2 4088.453} C_VEL
LIN {X 0,Y 535.97,Z 843.44,A -85,B 0,C 180,E1 4094.738,E2 4094.738} C_VEL
LIN {X 0,Y 536.034,Z 843.44,A -85,B 0,C 180,E1 4099.65,E2 4099.65} C_VEL
LIN {X 0,Y 536.001,Z 843.44,A -85,B 0,C 180,E1 4104.73,E2 4104.73} C_VEL
LIN {X 0,Y 536.03,Z 843.44,A -85,B 0,C 180,E1 4110.774,E2 4110.774} C_VEL
LIN {X 0,Y 536.188,Z 843.44,A -85,B 0,C 180,E1 4116.797,E2 4116.797} C_VEL
LIN {X 0,Y 536.354,Z 843.44,A -85,B 0,C 180,E1 4121.973,E2 4121.973} C_VEL
LIN {X 0,Y 536.493,Z 843.44,A -85,B 0,C 180,E1 4126.997,E2 4126.997} C_VEL
LIN {X 0,Y 536.408,Z 843.44,A -85,B 0,C 180,E1 4132.64,E2 4132.64} C_VEL
LIN {X 0,Y 536.403,Z 843.44,A -85,B 0,C 180,E1 4138.388,E2 4138.388} C_VEL
LIN {X 0,Y 536.464,Z 843.44,A -85,B 0,C 180,E1 4143.225,E2 4143.225} C_VEL
LIN {X 0,Y 536.345,Z 843.44,A -85,B 0,C 180,E1 4148.087,E2 4148.087} C_VEL
LIN {X 0,Y 536.305,Z 843.44,A -85,B 0,C 180,E1 4153.008,E2 4153.008} C_VEL
LIN {X 0,Y 536.258,Z 843.44,A -85,B 0,C 180,E1 4158.031,E2 4158.031} C_VEL
LIN {X 0,Y 536.188,Z 843.44,A -85,B 0,C 180,E1 4163.203,E2 4163.203} C_VEL
LIN {X 0,Y 536.162,Z 843.44,A -85,B 0,C 180,E1 4166.753,E2 4166.753} C_VEL
LIN {X 0,Y 533.634,Z 843.44,A -85,B 0,C 180,E1 4168.133,E2 4168.133} C_VEL
LIN {X 0,Y 528.157,Z 843.44,A -85,B 0,C 180,E1 4170.199,E2 4170.199} C_VEL
LIN {X 0,Y 528.07,Z 843.44,A -85,B 0,C 180,E1 4170.439,E2 4170.439} C_VEL
LIN {X 0,Y 528.147,Z 843.44,A -85,B 0,C 180,E1 4176.869,E2 4176.869} C_VEL
LIN {X 0,Y 528.089,Z 843.44,A -85,B 0,C 180,E1 4183.297,E2 4183.297} C_VEL
LIN {X 0,Y 528.055,Z 843.44,A -85,B 0,C 180,E1 4189.729,E2 4189.729} C_VEL
LIN {X 0,Y 528.092,Z 843.443,A -85,B 0,C 180,E1 4190.333,E2 4190.333} C_VEL
LIN {X 0,Y 532.551,Z 853.304,A -85,B 0,C 180,E1 4190.898,E2 4190.898} C_VEL
LIN {X 0,Y 544.039,Z 875.099,A -85,B 0,C 180,E1 4192.232,E2 4192.232} C_VEL
LIN {X 0,Y 543.031,Z 919.281,A -85,B 0,C 180,E1 4193.185,E2 4193.185} C_VEL
LIN {X 0,Y 541.157,Z 958.514,A -85,B 0,C 180,E1 4194.627,E2 4194.627} C_VEL
LIN {X 0,Y 538.745,Z 999.054,A -85,B 0,C 180,E1 4196.827,E2 4196.827} C_VEL
LIN {X 0,Y 536.13,Z 1037.17,A -85,B 0,C 180,E1 4199.664,E2 4199.664} C_VEL
LIN {X 0,Y 533.622,Z 1072.161,A -85,B 0,C 180,E1 4203.099,E2 4203.099} C_VEL
LIN {X 0,Y 531.58,Z 1102.34,A -85,B 0,C 180,E1 4206.935,E2 4206.935} C_VEL
LIN {X 0,Y 530.226,Z 1127.637,A -85,B 0,C 180,E1 4211.111,E2 4211.111} C_VEL
LIN {X 0,Y 529.429,Z 1147.673,A -85,B 0,C 180,E1 4215.508,E2 4215.508} C_VEL
LIN {X 0,Y 528.901,Z 1162.53,A -85,B 0,C 180,E1 4220.143,E2 4220.143} C_VEL
LIN {X 0,Y 528.738,Z 1170.731,A -85,B 0,C 180,E1 4224.267,E2 4224.267} C_VEL
LIN {X 0,Y 528.692,Z 1174.659,A -85,B 0,C 180,E1 4228.365,E2 4228.365} C_VEL
LIN {X 0,Y 528.879,Z 1173.792,A -85,B 0,C 180,E1 4233.039,E2 4233.039} C_VEL
LIN {X 0,Y 528.901,Z 1167.964,A -85,B 0,C 180,E1 4237.377,E2 4237.377} C_VEL
LIN {X 0,Y 529.113,Z 1156.566,A -85,B 0,C 180,E1 4241.933,E2 4241.933} C_VEL
LIN {X 0,Y 529.658,Z 1140.957,A -85,B 0,C 180,E1 4246.128,E2 4246.128} C_VEL
LIN {X 0,Y 530.771,Z 1117.692,A -85,B 0,C 180,E1 4250.671,E2 4250.671} C_VEL
LIN {X 0,Y 532.392,Z 1090.005,A -85,B 0,C 180,E1 4254.759,E2 4254.759} C_VEL
LIN {X 0,Y 534.645,Z 1057.634,A -85,B 0,C 180,E1 4258.444,E2 4258.444} C_VEL
LIN {X 0,Y 537.289,Z 1020.798,A -85,B 0,C 180,E1 4261.657,E2 4261.657} C_VEL
LIN {X 0,Y 539.876,Z 981.906,A -85,B 0,C 180,E1 4264.198,E2 4264.198} C_VEL
LIN {X 0,Y 542.194,Z 940.555,A -85,B 0,C 180,E1 4266.112,E2 4266.112} C_VEL
LIN {X 0,Y 543.817,Z 898.636,A -85,B 0,C 180,E1 4267.331,E2 4267.331} C_VEL
LIN {X 0,Y 543.731,Z 874.423,A -85,B 0,C 180,E1 4267.804,E2 4267.804} C_VEL
LIN {X 0,Y 528.213,Z 844.871,A -85,B 0,C 180,E1 4269.631,E2 4269.631} C_VEL
LIN {X 0,Y 528.075,Z 843.44,A -85,B 0,C 180,E1 4269.716,E2 4269.716} C_VEL
LIN {X 0,Y 528.087,Z 843.44,A -85,B 0,C 180,E1 4275.592,E2 4275.592} C_VEL
LIN {X 0,Y 528.123,Z 843.44,A -85,B 0,C 180,E1 4281.054,E2 4281.054} C_VEL
LIN {X 0,Y 528.101,Z 843.44,A -85,B 0,C 180,E1 4287.119,E2 4287.119} C_VEL
LIN {X 0,Y 528.172,Z 843.44,A -85,B 0,C 180,E1 4292.799,E2 4292.799} C_VEL
LIN {X 0,Y 528.338,Z 843.44,A -85,B 0,C 180,E1 4298.205,E2 4298.205} C_VEL
LIN {X 0,Y 528.438,Z 843.44,A -85,B 0,C 180,E1 4303.408,E2 4303.408} C_VEL
LIN {X 0,Y 528.478,Z 843.44,A -85,B 0,C 180,E1 4310.135,E2 4310.135} C_VEL
LIN {X 0,Y 528.641,Z 843.44,A -85,B 0,C 180,E1 4315.087,E2 4315.087} C_VEL
LIN {X 0,Y 528.642,Z 843.44,A -85,B 0,C 180,E1 4320,E2 4320} C_VEL
LIN {X 0,Y 528.614,Z 843.44,A -85,B 0,C 180,E1 4324.912,E2 4324.912} C_VEL
LIN {X 0,Y 528.52,Z 843.44,A -85,B 0,C 180,E1 4329.863,E2 4329.863} C_VEL
LIN {X 0,Y 528.461,Z 843.44,A -85,B 0,C 180,E1 4334.891,E2 4334.891} C_VEL
LIN {X 0,Y 528.379,Z 843.44,A -85,B 0,C 180,E1 4340.041,E2 4340.041} C_VEL
LIN {X 0,Y 528.202,Z 843.44,A -85,B 0,C 180,E1 4345.373,E2 4345.373} C_VEL
LIN {X 0,Y 528.221,Z 843.44,A -85,B 0,C 180,E1 4351.014,E2 4351.014} C_VEL
LIN {X 0,Y 528.331,Z 843.44,A -85,B 0,C 180,E1 4354.835,E2 4354.835} C_VEL
LIN {X 0,Y 528.034,Z 843.44,A -85,B 0,C 180,E1 4361.092,E2 4361.092} C_VEL
LIN {X 0,Y 528.011,Z 843.44,A -85,B 0,C 180,E1 4366.693,E2 4366.693} C_VEL
LIN {X 0,Y 528.242,Z 843.972,A -85,B 0,C 180,E1 4370.828,E2 4370.828} C_VEL
LIN {X 0,Y 543.504,Z 875.154,A -85,B 0,C 180,E1 4372.765,E2 4372.765} C_VEL
LIN {X 0,Y 541.946,Z 914.798,A -85,B 0,C 180,E1 4374.011,E2 4374.011} C_VEL
LIN {X 0,Y 539.799,Z 954.442,A -85,B 0,C 180,E1 4375.907,E2 4375.907} C_VEL
LIN {X 0,Y 537.17,Z 993.236,A -85,B 0,C 180,E1 4378.484,E2 4378.484} C_VEL
LIN {X 0,Y 534.497,Z 1030.237,A -85,B 0,C 180,E1 4381.778,E2 4381.778} C_VEL
LIN {X 0,Y 532.232,Z 1062.048,A -85,B 0,C 180,E1 4385.466,E2 4385.466} C_VEL
LIN {X 0,Y 530.589,Z 1089.289,A -85,B 0,C 180,E1 4389.557,E2 4389.557} C_VEL
LIN {X 0,Y 529.552,Z 1111.146,A -85,B 0,C 180,E1 4393.869,E2 4393.869} C_VEL
LIN {X 0,Y 529.082,Z 1128.041,A -85,B 0,C 180,E1 4398.483,E2 4398.483} C_VEL
LIN {X 0,Y 528.881,Z 1138.049,A -85,B 0,C 180,E1 4402.623,E2 4402.623} C_VEL
LIN {X 0,Y 528.826,Z 1143.673,A -85,B 0,C 180,E1 4406.728,E2 4406.728} C_VEL
LIN {X 0,Y 528.9,Z 1144.637,A -85,B 0,C 180,E1 4411.635,E2 4411.635} C_VEL
LIN {X 0,Y 528.831,Z 1140.665,A -85,B 0,C 180,E1 4415.732,E2 4415.732} C_VEL
LIN {X 0,Y 528.946,Z 1132.406,A -85,B 0,C 180,E1 4419.856,E2 4419.856} C_VEL
LIN {X 0,Y 529.324,Z 1117.571,A -85,B 0,C 180,E1 4424.478,E2 4424.478} C_VEL
LIN {X 0,Y 530.043,Z 1098.503,A -85,B 0,C 180,E1 4428.68,E2 4428.68} C_VEL
LIN {X 0,Y 531.454,Z 1074.39,A -85,B 0,C 180,E1 4432.717,E2 4432.717} C_VEL
LIN {X 0,Y 533.398,Z 1045.608,A -85,B 0,C 180,E1 4436.46,E2 4436.46} C_VEL
LIN {X 0,Y 535.787,Z 1012.241,A -85,B 0,C 180,E1 4439.843,E2 4439.843} C_VEL
LIN {X 0,Y 538.368,Z 975.89,A -85,B 0,C 180,E1 4442.672,E2 4442.672} C_VEL
LIN {X 0,Y 540.814,Z 938.406,A -85,B 0,C 180,E1 4444.853,E2 4444.853} C_VEL
LIN {X 0,Y 542.762,Z 898.061,A -85,B 0,C 180,E1 4446.498,E2 4446.498} C_VEL
LIN {X 0,Y 543.277,Z 874.721,A -85,B 0,C 180,E1 4447.175,E2 4447.175} C_VEL
LIN {X 0,Y 528.11,Z 844.452,A -85,B 0,C 180,E1 4449.086,E2 4449.086} C_VEL
LIN {X 0,Y 528.041,Z 843.44,A -85,B 0,C 180,E1 4449.218,E2 4449.218} C_VEL
LIN {X 0,Y 528.084,Z 843.44,A -85,B 0,C 180,E1 4455.592,E2 4455.592} C_VEL
LIN {X 0,Y 528.108,Z 843.44,A -85,B 0,C 180,E1 4461.053,E2 4461.053} C_VEL
LIN {X 0,Y 528.075,Z 843.44,A -85,B 0,C 180,E1 4467.118,E2 4467.118} C_VEL
LIN {X 0,Y 528.146,Z 843.44,A -85,B 0,C 180,E1 4472.798,E2 4472.798} C_VEL
LIN {X 0,Y 528.351,Z 843.44,A -85,B 0,C 180,E1 4478.206,E2 4478.206} C_VEL
LIN {X 0,Y 528.47,Z 843.44,A -85,B 0,C 180,E1 4483.41,E2 4483.41} C_VEL
LIN {X 0,Y 528.475,Z 843.44,A -85,B 0,C 180,E1 4488.471,E2 4488.471} C_VEL
LIN {X 0,Y 528.54,Z 843.44,A -85,B 0,C 180,E1 4493.443,E2 4493.443} C_VEL
LIN {X 0,Y 528.516,Z 843.44,A -85,B 0,C 180,E1 4498.364,E2 4498.364} C_VEL
LIN {X 0,Y 528.574,Z 843.44,A -85,B 0,C 180,E1 4503.273,E2 4503.273} C_VEL
LIN {X 0,Y 528.448,Z 843.44,A -85,B 0,C 180,E1 4508.208,E2 4508.208} C_VEL
LIN {X 0,Y 528.348,Z 843.44,A -85,B 0,C 180,E1 4513.815,E2 4513.815} C_VEL
LIN {X 0,Y 528.37,Z 843.44,A -85,B 0,C 180,E1 4519.529,E2 4519.529} C_VEL
LIN {X 0,Y 528.253,Z 843.44,A -85,B 0,C 180,E1 4525.371,E2 4525.371} C_VEL
LIN {X 0,Y 528.07,Z 843.44,A -85,B 0,C 180,E1 4530.439,E2 4530.439} C_VEL
LIN {X 0,Y 525.567,Z 843.44,A -85,B 0,C 180,E1 4531.841,E2 4531.841} C_VEL
LIN {X 0,Y 520.17,Z 843.44,A -85,B 0,C 180,E1 4533.942,E2 4533.942} C_VEL
LIN {X 0,Y 520.065,Z 843.44,A -85,B 0,C 180,E1 4534.185,E2 4534.185} C_VEL
LIN {X 0,Y 520.216,Z 843.44,A -85,B 0,C 180,E1 4539.653,E2 4539.653} C_VEL
LIN {X 0,Y 520.123,Z 843.44,A -85,B 0,C 180,E1 4545.869,E2 4545.869} C_VEL
LIN {X 0,Y 520.138,Z 843.535,A -85,B 0,C 180,E1 4549.607,E2 4549.607} C_VEL
LIN {X 0,Y 524.543,Z 853.112,A -85,B 0,C 180,E1 4550.18,E2 4550.18} C_VEL
LIN {X 0,Y 537.832,Z 878.485,A -85,B 0,C 180,E1 4551.774,E2 4551.774} C_VEL
LIN {X 0,Y 536.557,Z 922.178,A -85,B 0,C 180,E1 4552.759,E2 4552.759} C_VEL
LIN {X 0,Y 534.425,Z 962.518,A -85,B 0,C 180,E1 4554.319,E2 4554.319} C_VEL
LIN {X 0,Y 531.719,Z 1001.746,A -85,B 0,C 180,E1 4556.524,E2 4556.524} C_VEL
LIN {X 0,Y 528.975,Z 1038.565,A -85,B 0,C 180,E1 4559.341,E2 4559.341} C_VEL
LIN {X 0,Y 526.302,Z 1072.404,A -85,B 0,C 180,E1 4562.723,E2 4562.723} C_VEL
LIN {X 0,Y 524.087,Z 1101.882,A -85,B 0,C 180,E1 4566.516,E2 4566.516} C_VEL
LIN {X 0,Y 522.521,Z 1127.639,A -85,B 0,C 180,E1 4570.822,E2 4570.822} C_VEL
LIN {X 0,Y 521.598,Z 1147.408,A -85,B 0,C 180,E1 4575.212,E2 4575.212} C_VEL
LIN {X 0,Y 521.046,Z 1162.529,A -85,B 0,C 180,E1 4579.993,E2 4579.993} C_VEL
LIN {X 0,Y 520.845,Z 1170.731,A -85,B 0,C 180,E1 4584.18,E2 4584.18} C_VEL
LIN {X 0,Y 520.809,Z 1174.659,A -85,B 0,C 180,E1 4588.34,E2 4588.34} C_VEL
LIN {X 0,Y 521.055,Z 1174.659,A -85,B 0,C 180,E1 4591.66,E2 4591.66} C_VEL
LIN {X 0,Y 520.929,Z 1169.517,A -85,B 0,C 180,E1 4596.654,E2 4596.654} C_VEL
LIN {X 0,Y 521.215,Z 1159.205,A -85,B 0,C 180,E1 4601.227,E2 4601.227} C_VEL
LIN {X 0,Y 521.78,Z 1142.712,A -85,B 0,C 180,E1 4605.947,E2 4605.947} C_VEL
LIN {X 0,Y 522.843,Z 1121.767,A -85,B 0,C 180,E1 4610.264,E2 4610.264} C_VEL
LIN {X 0,Y 524.506,Z 1096.271,A -85,B 0,C 180,E1 4614.277,E2 4614.277} C_VEL
LIN {X 0,Y 526.77,Z 1066.104,A -85,B 0,C 180,E1 4617.975,E2 4617.975} C_VEL
LIN {X 0,Y 529.476,Z 1031.763,A -85,B 0,C 180,E1 4621.243,E2 4621.243} C_VEL
LIN {X 0,Y 532.383,Z 993.015,A -85,B 0,C 180,E1 4624.033,E2 4624.033} C_VEL
LIN {X 0,Y 535.032,Z 952.258,A -85,B 0,C 180,E1 4626.147,E2 4626.147} C_VEL
LIN {X 0,Y 537.125,Z 909.056,A -85,B 0,C 180,E1 4627.607,E2 4627.607} C_VEL
LIN {X 0,Y 537.535,Z 877.337,A -85,B 0,C 180,E1 4628.27,E2 4628.27} C_VEL
LIN {X 0,Y 520.289,Z 844.923,A -85,B 0,C 180,E1 4630.355,E2 4630.355} C_VEL
LIN {X 0,Y 520.138,Z 843.44,A -85,B 0,C 180,E1 4630.453,E2 4630.453} C_VEL
LIN {X 0,Y 520.168,Z 843.44,A -85,B 0,C 180,E1 4636.49,E2 4636.49} C_VEL
LIN {X 0,Y 520.166,Z 843.44,A -85,B 0,C 180,E1 4642.469,E2 4642.469} C_VEL
LIN {X 0,Y 520.193,Z 843.44,A -85,B 0,C 180,E1 4648.524,E2 4648.524} C_VEL
LIN {X 0,Y 520.281,Z 843.44,A -85,B 0,C 180,E1 4654.212,E2 4654.212} C_VEL
LIN {X 0,Y 520.459,Z 843.44,A -85,B 0,C 180,E1 4659.64,E2 4659.64} C_VEL
LIN {X 0,Y 520.37,Z 843.44,A -85,B 0,C 180,E1 4664.872,E2 4664.872} C_VEL
LIN {X 0,Y 520.593,Z 843.44,A -85,B 0,C 180,E1 4670.245,E2 4670.245} C_VEL
LIN {X 0,Y 520.733,Z 843.44,A -85,B 0,C 180,E1 4675.013,E2 4675.013} C_VEL
LIN {X 0,Y 520.754,Z 843.44,A -85,B 0,C 180,E1 4680,E2 4680} C_VEL
LIN {X 0,Y 520.701,Z 843.44,A -85,B 0,C 180,E1 4684.987,E2 4684.987} C_VEL
LIN {X 0,Y 520.623,Z 843.44,A -85,B 0,C 180,E1 4690.015,E2 4690.015} C_VEL
LIN {X 0,Y 520.526,Z 843.44,A -85,B 0,C 180,E1 4695.123,E2 4695.123} C_VEL
